LIN {X 0,Y 516.172,Z 433.767,A -85,B 0,C 180,E1 -4909.681,E2 -4909.681} C_VEL
LIN {X 0,Y 516.191,Z 433.561,A -85,B 0,C 180,E1 -4910.899,E2 -4910.899} C_VEL
LIN {X 0,Y 516.175,Z 431.928,A -85,B 0,C 180,E1 -4912.214,E2 -4912.214} C_VEL
LIN {X 0,Y 516.288,Z 429.068,A -85,B 0,C 180,E1 -4913.429,E2 -4913.429} C_VEL
LIN {X 0,Y 516.355,Z 425.479,A -85,B 0,C 180,E1 -4914.491,E2 -4914.491} C_VEL
LIN {X 0,Y 516.462,Z 420.419,A -85,B 0,C 180,E1 -4915.616,E2 -4915.616} C_VEL
LIN {X 0,Y 516.626,Z 413.305,A -85,B 0,C 180,E1 -4916.803,E2 -4916.803} C_VEL
LIN {X 0,Y 516.784,Z 406.191,A -85,B 0,C 180,E1 -4917.726,E2 -4917.726} C_VEL
LIN {X 0,Y 516.968,Z 399.489,A -85,B 0,C 180,E1 -4918.439,E2 -4918.439} C_VEL
LIN {X 0,Y 517.059,Z 393.49,A -85,B 0,C 180,E1 -4918.98,E2 -4918.98} C_VEL
LIN {X 0,Y 517.216,Z 385.286,A -85,B 0,C 180,E1 -4919.591,E2 -4919.591} C_VEL
LIN {X 0,Y 517.396,Z 376.875,A -85,B 0,C 180,E1 -4920.093,E2 -4920.093} C_VEL
LIN {X 0,Y 517.533,Z 368.879,A -85,B 0,C 180,E1 -4920.47,E2 -4920.47} C_VEL
LIN {X 0,Y 517.4,Z 363.16,A -85,B 0,C 180,E1 -4920.698,E2 -4920.698} C_VEL
LIN {X 0,Y 516.294,Z 355.849,A -85,B 0,C 180,E1 -4920.963,E2 -4920.963} C_VEL
LIN {X 0,Y 516.339,Z 351.268,A -85,B 0,C 180,E1 -4924.178,E2 -4924.178} C_VEL
LIN {X 0,Y 516.335,Z 347.701,A -85,B 0,C 180,E1 -4926.75,E2 -4926.75} C_VEL
LIN {X 0,Y 516.376,Z 343.028,A -85,B 0,C 180,E1 -4930.107,E2 -4930.107} C_VEL
LIN {X 0,Y 516.437,Z 339.664,A -85,B 0,C 180,E1 -4932.578,E2 -4932.578} C_VEL
LIN {X 0,Y 516.461,Z 335.27,A -85,B 0,C 180,E1 -4935.821,E2 -4935.821} C_VEL
LIN {X 0,Y 516.631,Z 330.958,A -85,B 0,C 180,E1 -4939.02,E2 -4939.02} C_VEL
LIN {X 0,Y 516.634,Z 328.948,A -85,B 0,C 180,E1 -4940.604,E2 -4940.604} C_VEL
LIN {X 0,Y 517.004,Z 328.898,A -85,B 0,C 180,E1 -4942.972,E2 -4942.972} C_VEL
LIN {X 0,Y 516.928,Z 328.907,A -85,B 0,C 180,E1 -4945.32,E2 -4945.32} C_VEL
LIN {X 0,Y 517.072,Z 328.89,A -85,B 0,C 180,E1 -4947.662,E2 -4947.662} C_VEL
LIN {X 0,Y 517.085,Z 328.89,A -85,B 0,C 180,E1 -4950.778,E2 -4950.778} C_VEL
LIN {X 0,Y 517.006,Z 328.899,A -85,B 0,C 180,E1 -4953.116,E2 -4953.116} C_VEL
LIN {X 0,Y 517,Z 328.899,A -85,B 0,C 180,E1 -4956.242,E2 -4956.242} C_VEL
LIN {X 0,Y 516.948,Z 328.907,A -85,B 0,C 180,E1 -4959.388,E2 -4959.388} C_VEL
LIN {X 0,Y 516.971,Z 328.905,A -85,B 0,C 180,E1 -4961.823,E2 -4961.823} C_VEL
LIN {X 0,Y 516.931,Z 328.907,A -85,B 0,C 180,E1 -4965.146,E2 -4965.146} C_VEL
LIN {X 0,Y 516.913,Z 328.909,A -85,B 0,C 180,E1 -4968.221,E2 -4968.221} C_VEL
LIN {X 0,Y 516.9,Z 328.911,A -85,B 0,C 180,E1 -4970.701,E2 -4970.701} C_VEL
LIN {X 0,Y 516.897,Z 328.912,A -85,B 0,C 180,E1 -4974.071,E2 -4974.071} C_VEL
LIN {X 0,Y 516.915,Z 328.91,A -85,B 0,C 180,E1 -4976.657,E2 -4976.657} C_VEL
LIN {X 0,Y 516.91,Z 328.911,A -85,B 0,C 180,E1 -4979.526,E2 -4979.526} C_VEL
LIN {X 0,Y 516.887,Z 328.914,A -85,B 0,C 180,E1 -4982.544,E2 -4982.544} C_VEL
LIN {X 0,Y 516.87,Z 328.915,A -85,B 0,C 180,E1 -4985.332,E2 -4985.332} C_VEL
LIN {X 0,Y 516.87,Z 328.915,A -85,B 0,C 180,E1 -4987.944,E2 -4987.944} C_VEL
LIN {X 0,Y 516.893,Z 328.913,A -85,B 0,C 180,E1 -4990.739,E2 -4990.739} C_VEL
LIN {X 0,Y 516.868,Z 328.914,A -85,B 0,C 180,E1 -4993.903,E2 -4993.903} C_VEL
LIN {X 0,Y 516.867,Z 328.915,A -85,B 0,C 180,E1 -4996.107,E2 -4996.107} C_VEL
LIN {X 0,Y 516.889,Z 328.915,A -85,B 0,C 180,E1 -4999.26,E2 -4999.26} C_VEL
LIN {X 0,Y 516.871,Z 328.916,A -85,B 0,C 180,E1 -5002.056,E2 -5002.056} C_VEL
LIN {X 0,Y 516.882,Z 328.915,A -85,B 0,C 180,E1 -5005.177,E2 -5005.177} C_VEL
LIN {X 0,Y 516.869,Z 328.917,A -85,B 0,C 180,E1 -5007.976,E2 -5007.976} C_VEL
LIN {X 0,Y 516.922,Z 328.909,A -85,B 0,C 180,E1 -5010.697,E2 -5010.697} C_VEL
LIN {X 0,Y 516.928,Z 328.908,A -85,B 0,C 180,E1 -5013.804,E2 -5013.804} C_VEL
LIN {X 0,Y 516.885,Z 328.913,A -85,B 0,C 180,E1 -5016.778,E2 -5016.778} C_VEL
LIN {X 0,Y 516.926,Z 328.907,A -85,B 0,C 180,E1 -5019.732,E2 -5019.732} C_VEL
LIN {X 0,Y 516.918,Z 328.91,A -85,B 0,C 180,E1 -5022.597,E2 -5022.597} C_VEL
LIN {X 0,Y 516.928,Z 328.908,A -85,B 0,C 180,E1 -5025.031,E2 -5025.031} C_VEL
LIN {X 0,Y 516.991,Z 328.901,A -85,B 0,C 180,E1 -5028.235,E2 -5028.235} C_VEL
LIN {X 0,Y 516.96,Z 328.904,A -85,B 0,C 180,E1 -5031.4,E2 -5031.4} C_VEL
LIN {X 0,Y 517,Z 328.9,A -85,B 0,C 180,E1 -5033.758,E2 -5033.758} C_VEL
LIN {X 0,Y 517.076,Z 328.889,A -85,B 0,C 180,E1 -5037.664,E2 -5037.664} C_VEL
LIN {X 0,Y 517.087,Z 328.889,A -85,B 0,C 180,E1 -5040.78,E2 -5040.78} C_VEL
LIN {X 0,Y 517.007,Z 328.899,A -85,B 0,C 180,E1 -5043.118,E2 -5043.118} C_VEL
LIN {X 0,Y 517,Z 328.899,A -85,B 0,C 180,E1 -5046.244,E2 -5046.244} C_VEL
LIN {X 0,Y 516.945,Z 328.907,A -85,B 0,C 180,E1 -5049.39,E2 -5049.39} C_VEL
LIN {X 0,Y 516.973,Z 328.903,A -85,B 0,C 180,E1 -5051.825,E2 -5051.825} C_VEL
LIN {X 0,Y 516.934,Z 328.908,A -85,B 0,C 180,E1 -5055.147,E2 -5055.147} C_VEL
LIN {X 0,Y 516.917,Z 328.908,A -85,B 0,C 180,E1 -5058.223,E2 -5058.223} C_VEL
LIN {X 0,Y 516.903,Z 328.91,A -85,B 0,C 180,E1 -5060.702,E2 -5060.702} C_VEL
LIN {X 0,Y 516.903,Z 328.91,A -85,B 0,C 180,E1 -5064.073,E2 -5064.073} C_VEL
LIN {X 0,Y 516.921,Z 328.908,A -85,B 0,C 180,E1 -5066.659,E2 -5066.659} C_VEL
LIN {X 0,Y 516.917,Z 328.91,A -85,B 0,C 180,E1 -5069.528,E2 -5069.528} C_VEL
LIN {X 0,Y 516.89,Z 328.913,A -85,B 0,C 180,E1 -5072.545,E2 -5072.545} C_VEL
LIN {X 0,Y 516.877,Z 328.914,A -85,B 0,C 180,E1 -5075.334,E2 -5075.334} C_VEL
LIN {X 0,Y 516.875,Z 328.914,A -85,B 0,C 180,E1 -5077.945,E2 -5077.945} C_VEL
LIN {X 0,Y 516.879,Z 328.916,A -85,B 0,C 180,E1 -5080.743,E2 -5080.743} C_VEL
LIN {X 0,Y 516.898,Z 328.912,A -85,B 0,C 180,E1 -5082.83,E2 -5082.83} C_VEL
LIN {X 0,Y 516.917,Z 328.909,A -85,B 0,C 180,E1 -5085.011,E2 -5085.011} C_VEL
LIN {X 0,Y 516.912,Z 328.91,A -85,B 0,C 180,E1 -5088.399,E2 -5088.399} C_VEL
LIN {X 0,Y 516.878,Z 328.914,A -85,B 0,C 180,E1 -5091.286,E2 -5091.286} C_VEL
LIN {X 0,Y 516.912,Z 328.911,A -85,B 0,C 180,E1 -5094.664,E2 -5094.664} C_VEL
LIN {X 0,Y 516.971,Z 329.042,A -85,B 0,C 180,E1 -5095.089,E2 -5095.089} C_VEL
LIN {X 0,Y 517.728,Z 334.233,A -85,B 0,C 180,E1 -5097.114,E2 -5097.114} C_VEL
LIN {X 0,Y 517.54,Z 340.461,A -85,B 0,C 180,E1 -5099.389,E2 -5099.389} C_VEL
LIN {X 0,Y 517.319,Z 347.853,A -85,B 0,C 180,E1 -5102.013,E2 -5102.013} C_VEL
LIN {X 0,Y 517.105,Z 355.534,A -85,B 0,C 180,E1 -5104.653,E2 -5104.653} C_VEL
LIN {X 0,Y 516.938,Z 363.131,A -85,B 0,C 180,E1 -5107.205,E2 -5107.205} C_VEL
LIN {X 0,Y 516.741,Z 373.276,A -85,B 0,C 180,E1 -5110.537,E2 -5110.537} C_VEL
LIN {X 0,Y 516.594,Z 382.323,A -85,B 0,C 180,E1 -5113.401,E2 -5113.401} C_VEL
LIN {X 0,Y 516.522,Z 390.164,A -85,B 0,C 180,E1 -5115.824,E2 -5115.824} C_VEL
LIN {X 0,Y 516.441,Z 398.672,A -85,B 0,C 180,E1 -5118.469,E2 -5118.469} C_VEL
LIN {X 0,Y 516.417,Z 400.594,A -85,B 0,C 180,E1 -5119.042,E2 -5119.042} C_VEL
LIN {X 0,Y 517.546,Z 412.161,A -85,B 0,C 180,E1 -5119.388,E2 -5119.388} C_VEL
LIN {X 0,Y 517.385,Z 422.491,A -85,B 0,C 180,E1 -5119.83,E2 -5119.83} C_VEL
LIN {X 0,Y 517.179,Z 431.229,A -85,B 0,C 180,E1 -5120.32,E2 -5120.32} C_VEL
LIN {X 0,Y 517.022,Z 439.578,A -85,B 0,C 180,E1 -5120.909,E2 -5120.909} C_VEL
LIN {X 0,Y 516.818,Z 447.479,A -85,B 0,C 180,E1 -5121.595,E2 -5121.595} C_VEL
LIN {X 0,Y 516.672,Z 454.871,A -85,B 0,C 180,E1 -5122.38,E2 -5122.38} C_VEL
LIN {X 0,Y 516.533,Z 462.212,A -85,B 0,C 180,E1 -5123.337,E2 -5123.337} C_VEL
LIN {X 0,Y 516.448,Z 468.264,A -85,B 0,C 180,E1 -5124.339,E2 -5124.339} C_VEL
LIN {X 0,Y 516.314,Z 472.898,A -85,B 0,C 180,E1 -5125.316,E2 -5125.316} C_VEL
LIN {X 0,Y 516.364,Z 475.915,A -85,B 0,C 180,E1 -5126.099,E2 -5126.099} C_VEL
LIN {X 0,Y 516.294,Z 478.248,A -85,B 0,C 180,E1 -5126.88,E2 -5126.88} C_VEL
LIN {X 0,Y 516.263,Z 480.005,A -85,B 0,C 180,E1 -5127.66,E2 -5127.66} C_VEL
LIN {X 0,Y 516.191,Z 481.261,A -85,B 0,C 180,E1 -5128.441,E2 -5128.441} C_VEL
LIN {X 0,Y 516.158,Z 482.041,A -85,B 0,C 180,E1 -5129.221,E2 -5129.221} C_VEL
LIN {X 0,Y 516.156,Z 482.335,A -85,B 0,C 180,E1 -5130.001,E2 -5130.001} C_VEL
LIN {X 0,Y 516.158,Z 482.036,A -85,B 0,C 180,E1 -5130.781,E2 -5130.781} C_VEL
LIN {X 0,Y 516.191,Z 481.25,A -85,B 0,C 180,E1 -5131.561,E2 -5131.561} C_VEL
LIN {X 0,Y 516.263,Z 479.988,A -85,B 0,C 180,E1 -5132.342,E2 -5132.342} C_VEL
LIN {X 0,Y 516.323,Z 477.065,A -85,B 0,C 180,E1 -5133.513,E2 -5133.513} C_VEL
LIN {X 0,Y 516.342,Z 474.398,A -85,B 0,C 180,E1 -5134.294,E2 -5134.294} C_VEL
LIN {X 0,Y 516.425,Z 469.184,A -85,B 0,C 180,E1 -5135.467,E2 -5135.467} C_VEL
LIN {X 0,Y 516.516,Z 463.713,A -85,B 0,C 180,E1 -5136.423,E2 -5136.423} C_VEL
LIN {X 0,Y 516.633,Z 456.509,A -85,B 0,C 180,E1 -5137.426,E2 -5137.426} C_VEL
LIN {X 0,Y 516.797,Z 448.426,A -85,B 0,C 180,E1 -5138.309,E2 -5138.309} C_VEL
LIN {X 0,Y 516.989,Z 440.714,A -85,B 0,C 180,E1 -5138.995,E2 -5138.995} C_VEL
LIN {X 0,Y 517.146,Z 432.616,A -85,B 0,C 180,E1 -5139.584,E2 -5139.584} C_VEL
LIN {X 0,Y 517.337,Z 424.231,A -85,B 0,C 180,E1 -5140.074,E2 -5140.074} C_VEL
LIN {X 0,Y 517.514,Z 415.677,A -85,B 0,C 180,E1 -5140.466,E2 -5140.466} C_VEL
LIN {X 0,Y 517.365,Z 408.802,A -85,B 0,C 180,E1 -5140.717,E2 -5140.717} C_VEL
LIN {X 0,Y 516.427,Z 400.26,A -85,B 0,C 180,E1 -5140.984,E2 -5140.984} C_VEL
LIN {X 0,Y 516.52,Z 389.965,A -85,B 0,C 180,E1 -5144.178,E2 -5144.178} C_VEL
LIN {X 0,Y 516.594,Z 380.776,A -85,B 0,C 180,E1 -5147.008,E2 -5147.008} C_VEL
LIN {X 0,Y 516.734,Z 373.032,A -85,B 0,C 180,E1 -5149.465,E2 -5149.465} C_VEL
LIN {X 0,Y 516.868,Z 364.07,A -85,B 0,C 180,E1 -5152.389,E2 -5152.389} C_VEL
LIN {X 0,Y 517.089,Z 355.16,A -85,B 0,C 180,E1 -5155.35,E2 -5155.35} C_VEL
LIN {X 0,Y 517.301,Z 346.385,A -85,B 0,C 180,E1 -5158.393,E2 -5158.393} C_VEL
LIN {X 0,Y 517.626,Z 338.595,A -85,B 0,C 180,E1 -5161.198,E2 -5161.198} C_VEL
LIN {X 0,Y 517.721,Z 334.128,A -85,B 0,C 180,E1 -5162.889,E2 -5162.889} C_VEL
LIN {X 0,Y 516.897,Z 328.913,A -85,B 0,C 180,E1 -5165.01,E2 -5165.01} C_VEL
LIN {X 0,Y 516.885,Z 328.915,A -85,B 0,C 180,E1 -5167.943,E2 -5167.943} C_VEL
LIN {X 0,Y 516.888,Z 328.918,A -85,B 0,C 180,E1 -5170.742,E2 -5170.742} C_VEL
LIN {X 0,Y 516.89,Z 328.918,A -85,B 0,C 180,E1 -5172.832,E2 -5172.832} C_VEL
LIN {X 0,Y 516.901,Z 328.915,A -85,B 0,C 180,E1 -5175.007,E2 -5175.007} C_VEL
LIN {X 0,Y 516.919,Z 328.91,A -85,B 0,C 180,E1 -5178.399,E2 -5178.399} C_VEL
LIN {X 0,Y 516.883,Z 328.915,A -85,B 0,C 180,E1 -5181.284,E2 -5181.284} C_VEL
LIN {X 0,Y 516.877,Z 328.914,A -85,B 0,C 180,E1 -5184.22,E2 -5184.22} C_VEL
LIN {X 0,Y 516.887,Z 328.915,A -85,B 0,C 180,E1 -5187.052,E2 -5187.052} C_VEL
LIN {X 0,Y 516.893,Z 328.912,A -85,B 0,C 180,E1 -5189.796,E2 -5189.796} C_VEL
LIN {X 0,Y 516.93,Z 328.907,A -85,B 0,C 180,E1 -5192.467,E2 -5192.467} C_VEL
LIN {X 0,Y 516.915,Z 328.911,A -85,B 0,C 180,E1 -5195.072,E2 -5195.072} C_VEL
LIN {X 0,Y 516.892,Z 328.912,A -85,B 0,C 180,E1 -5198.462,E2 -5198.462} C_VEL
LIN {X 0,Y 516.906,Z 328.912,A -85,B 0,C 180,E1 -5200.954,E2 -5200.954} C_VEL
LIN {X 0,Y 516.911,Z 328.911,A -85,B 0,C 180,E1 -5203.41,E2 -5203.41} C_VEL
LIN {X 0,Y 516.898,Z 328.914,A -85,B 0,C 180,E1 -5205.833,E2 -5205.833} C_VEL
LIN {X 0,Y 516.973,Z 328.905,A -85,B 0,C 180,E1 -5208.233,E2 -5208.233} C_VEL
LIN {X 0,Y 516.961,Z 328.904,A -85,B 0,C 180,E1 -5211.399,E2 -5211.399} C_VEL
LIN {X 0,Y 517.029,Z 328.896,A -85,B 0,C 180,E1 -5214.539,E2 -5214.539} C_VEL
LIN {X 0,Y 517.084,Z 328.891,A -85,B 0,C 180,E1 -5217.662,E2 -5217.662} C_VEL
LIN {X 0,Y 517.099,Z 328.886,A -85,B 0,C 180,E1 -5220.778,E2 -5220.778} C_VEL
LIN {X 0,Y 517.014,Z 328.897,A -85,B 0,C 180,E1 -5223.116,E2 -5223.116} C_VEL
LIN {X 0,Y 517.014,Z 328.898,A -85,B 0,C 180,E1 -5226.242,E2 -5226.242} C_VEL
LIN {X 0,Y 516.944,Z 328.908,A -85,B 0,C 180,E1 -5229.389,E2 -5229.389} C_VEL
LIN {X 0,Y 516.956,Z 328.907,A -85,B 0,C 180,E1 -5231.806,E2 -5231.806} C_VEL
LIN {X 0,Y 516.948,Z 328.908,A -85,B 0,C 180,E1 -5235.145,E2 -5235.145} C_VEL
LIN {X 0,Y 516.852,Z 328.921,A -85,B 0,C 180,E1 -5237.853,E2 -5237.853} C_VEL
LIN {X 0,Y 516.655,Z 328.945,A -85,B 0,C 180,E1 -5239.054,E2 -5239.054} C_VEL
LIN {X 0,Y 516.57,Z 332.084,A -85,B 0,C 180,E1 -5241.55,E2 -5241.55} C_VEL
LIN {X 0,Y 516.545,Z 335.708,A -85,B 0,C 180,E1 -5244.273,E2 -5244.273} C_VEL
LIN {X 0,Y 516.45,Z 338.912,A -85,B 0,C 180,E1 -5246.683,E2 -5246.683} C_VEL
LIN {X 0,Y 516.427,Z 342.589,A -85,B 0,C 180,E1 -5249.428,E2 -5249.428} C_VEL
LIN {X 0,Y 516.338,Z 346.763,A -85,B 0,C 180,E1 -5252.445,E2 -5252.445} C_VEL
LIN {X 0,Y 516.314,Z 350.521,A -85,B 0,C 180,E1 -5255.242,E2 -5255.242} C_VEL
LIN {X 0,Y 516.235,Z 354.157,A -85,B 0,C 180,E1 -5257.85,E2 -5257.85} C_VEL
LIN {X 0,Y 516.279,Z 356.115,A -85,B 0,C 180,E1 -5259.153,E2 -5259.153} C_VEL
LIN {X 0,Y 517.638,Z 366.34,A -85,B 0,C 180,E1 -5259.513,E2 -5259.513} C_VEL
LIN {X 0,Y 517.445,Z 375.523,A -85,B 0,C 180,E1 -5259.921,E2 -5259.921} C_VEL
LIN {X 0,Y 517.305,Z 383.809,A -85,B 0,C 180,E1 -5260.397,E2 -5260.397} C_VEL
LIN {X 0,Y 517.089,Z 391.927,A -85,B 0,C 180,E1 -5260.978,E2 -5260.978} C_VEL
LIN {X 0,Y 516.973,Z 399.12,A -85,B 0,C 180,E1 -5261.608,E2 -5261.608} C_VEL
LIN {X 0,Y 516.816,Z 405.767,A -85,B 0,C 180,E1 -5262.308,E2 -5262.308} C_VEL
LIN {X 0,Y 516.68,Z 411.965,A -85,B 0,C 180,E1 -5263.094,E2 -5263.094} C_VEL
LIN {X 0,Y 516.499,Z 418.569,A -85,B 0,C 180,E1 -5264.126,E2 -5264.126} C_VEL
LIN {X 0,Y 515.834,Z 421.674,A -85,B 0,C 180,E1 -5264.679,E2 -5264.679} C_VEL
LIN {X 0,Y 514.218,Z 424.431,A -85,B 0,C 180,E1 -5265.238,E2 -5265.238} C_VEL
LIN {X 0,Y 510.396,Z 428.868,A -85,B 0,C 180,E1 -5266.404,E2 -5266.404} C_VEL
LIN {X 0,Y 509.222,Z 430.843,A -85,B 0,C 180,E1 -5267.14,E2 -5267.14} C_VEL
LIN {X 0,Y 509.192,Z 431.048,A -85,B 0,C 180,E1 -5267.248,E2 -5267.248} C_VEL
LIN {X 0,Y 509.139,Z 433.208,A -85,B 0,C 180,E1 -5268.502,E2 -5268.502} C_VEL
LIN {X 0,Y 509.102,Z 434.048,A -85,B 0,C 180,E1 -5269.546,E2 -5269.546} C_VEL
LIN {X 0,Y 509.084,Z 434.009,A -85,B 0,C 180,E1 -5270.63,E2 -5270.63} C_VEL
LIN {X 0,Y 509.092,Z 432.825,A -85,B 0,C 180,E1 -5271.893,E2 -5271.893} C_VEL
LIN {X 0,Y 509.179,Z 430.248,A -85,B 0,C 180,E1 -5273.181,E2 -5273.181} C_VEL
LIN {X 0,Y 509.275,Z 427.574,A -85,B 0,C 180,E1 -5274.084,E2 -5274.084} C_VEL
LIN {X 0,Y 509.334,Z 422.599,A -85,B 0,C 180,E1 -5275.306,E2 -5275.306} C_VEL
LIN {X 0,Y 509.439,Z 418.025,A -85,B 0,C 180,E1 -5276.187,E2 -5276.187} C_VEL
LIN {X 0,Y 509.572,Z 413.446,A -85,B 0,C 180,E1 -5276.921,E2 -5276.921} C_VEL
LIN {X 0,Y 509.771,Z 406.566,A -85,B 0,C 180,E1 -5277.824,E2 -5277.824} C_VEL
LIN {X 0,Y 509.971,Z 399.395,A -85,B 0,C 180,E1 -5278.594,E2 -5278.594} C_VEL
LIN {X 0,Y 510.072,Z 392.071,A -85,B 0,C 180,E1 -5279.244,E2 -5279.244} C_VEL
LIN {X 0,Y 510.308,Z 382.77,A -85,B 0,C 180,E1 -5279.91,E2 -5279.91} C_VEL
LIN {X 0,Y 510.566,Z 371.407,A -85,B 0,C 180,E1 -5280.52,E2 -5280.52} C_VEL
LIN {X 0,Y 510.369,Z 363.419,A -85,B 0,C 180,E1 -5280.847,E2 -5280.847} C_VEL
LIN {X 0,Y 509.201,Z 356.154,A -85,B 0,C 180,E1 -5281.113,E2 -5281.113} C_VEL
LIN {X 0,Y 509.25,Z 352.367,A -85,B 0,C 180,E1 -5283.792,E2 -5283.792} C_VEL
LIN {X 0,Y 509.245,Z 348.725,A -85,B 0,C 180,E1 -5286.407,E2 -5286.407} C_VEL
LIN {X 0,Y 509.249,Z 345.203,A -85,B 0,C 180,E1 -5288.971,E2 -5288.971} C_VEL
LIN {X 0,Y 509.391,Z 340.63,A -85,B 0,C 180,E1 -5292.329,E2 -5292.329} C_VEL
LIN {X 0,Y 509.407,Z 336.179,A -85,B 0,C 180,E1 -5295.62,E2 -5295.62} C_VEL
LIN {X 0,Y 509.559,Z 331.841,A -85,B 0,C 180,E1 -5298.866,E2 -5298.866} C_VEL
LIN {X 0,Y 509.57,Z 329.827,A -85,B 0,C 180,E1 -5300.473,E2 -5300.473} C_VEL
LIN {X 0,Y 509.942,Z 329.778,A -85,B 0,C 180,E1 -5302.874,E2 -5302.874} C_VEL
LIN {X 0,Y 509.896,Z 329.783,A -85,B 0,C 180,E1 -5305.255,E2 -5305.255} C_VEL
LIN {X 0,Y 510.044,Z 329.766,A -85,B 0,C 180,E1 -5307.63,E2 -5307.63} C_VEL
LIN {X 0,Y 510.044,Z 329.766,A -85,B 0,C 180,E1 -5309.999,E2 -5309.999} C_VEL
LIN {X 0,Y 510.047,Z 329.765,A -85,B 0,C 180,E1 -5312.368,E2 -5312.368} C_VEL
LIN {X 0,Y 509.998,Z 329.772,A -85,B 0,C 180,E1 -5315.534,E2 -5315.534} C_VEL
LIN {X 0,Y 509.941,Z 329.78,A -85,B 0,C 180,E1 -5317.921,E2 -5317.921} C_VEL
LIN {X 0,Y 509.914,Z 329.781,A -85,B 0,C 180,E1 -5321.124,E2 -5321.124} C_VEL
LIN {X 0,Y 509.852,Z 329.789,A -85,B 0,C 180,E1 -5324.365,E2 -5324.365} C_VEL
LIN {X 0,Y 509.89,Z 329.786,A -85,B 0,C 180,E1 -5327.651,E2 -5327.651} C_VEL
LIN {X 0,Y 509.873,Z 329.787,A -85,B 0,C 180,E1 -5330.401,E2 -5330.401} C_VEL
LIN {X 0,Y 509.823,Z 329.794,A -85,B 0,C 180,E1 -5333.562,E2 -5333.562} C_VEL
LIN {X 0,Y 509.899,Z 329.784,A -85,B 0,C 180,E1 -5336.379,E2 -5336.379} C_VEL
LIN {X 0,Y 509.872,Z 329.789,A -85,B 0,C 180,E1 -5338.843,E2 -5338.843} C_VEL
LIN {X 0,Y 509.812,Z 329.794,A -85,B 0,C 180,E1 -5341.589,E2 -5341.589} C_VEL
LIN {X 0,Y 509.84,Z 329.79,A -85,B 0,C 180,E1 -5344.413,E2 -5344.413} C_VEL
LIN {X 0,Y 509.808,Z 329.797,A -85,B 0,C 180,E1 -5347.34,E2 -5347.34} C_VEL
LIN {X 0,Y 509.848,Z 329.789,A -85,B 0,C 180,E1 -5350.38,E2 -5350.38} C_VEL
LIN {X 0,Y 509.826,Z 329.794,A -85,B 0,C 180,E1 -5353.064,E2 -5353.064} C_VEL
LIN {X 0,Y 509.815,Z 329.795,A -85,B 0,C 180,E1 -5355.792,E2 -5355.792} C_VEL
LIN {X 0,Y 509.85,Z 329.79,A -85,B 0,C 180,E1 -5358.576,E2 -5358.576} C_VEL
LIN {X 0,Y 509.843,Z 329.791,A -85,B 0,C 180,E1 -5361.785,E2 -5361.785} C_VEL
LIN {X 0,Y 509.833,Z 329.792,A -85,B 0,C 180,E1 -5364.624,E2 -5364.624} C_VEL
LIN {X 0,Y 509.852,Z 329.789,A -85,B 0,C 180,E1 -5367.482,E2 -5367.482} C_VEL
LIN {X 0,Y 509.867,Z 329.789,A -85,B 0,C 180,E1 -5370.269,E2 -5370.269} C_VEL
LIN {X 0,Y 509.871,Z 329.788,A -85,B 0,C 180,E1 -5372.945,E2 -5372.945} C_VEL
LIN {X 0,Y 509.875,Z 329.786,A -85,B 0,C 180,E1 -5375.575,E2 -5375.575} C_VEL
LIN {X 0,Y 509.836,Z 329.791,A -85,B 0,C 180,E1 -5378.15,E2 -5378.15} C_VEL
LIN {X 0,Y 509.852,Z 329.789,A -85,B 0,C 180,E1 -5380.682,E2 -5380.682} C_VEL
LIN {X 0,Y 509.875,Z 329.786,A -85,B 0,C 180,E1 -5383.175,E2 -5383.175} C_VEL
LIN {X 0,Y 509.851,Z 329.788,A -85,B 0,C 180,E1 -5385.635,E2 -5385.635} C_VEL
LIN {X 0,Y 509.91,Z 329.781,A -85,B 0,C 180,E1 -5388.875,E2 -5388.875} C_VEL
LIN {X 0,Y 509.94,Z 329.78,A -85,B 0,C 180,E1 -5392.079,E2 -5392.079} C_VEL
LIN {X 0,Y 509.973,Z 329.777,A -85,B 0,C 180,E1 -5394.465,E2 -5394.465} C_VEL
LIN {X 0,Y 510.047,Z 329.765,A -85,B 0,C 180,E1 -5397.632,E2 -5397.632} C_VEL
LIN {X 0,Y 510.056,Z 329.764,A -85,B 0,C 180,E1 -5400.79,E2 -5400.79} C_VEL
LIN {X 0,Y 509.95,Z 329.778,A -85,B 0,C 180,E1 -5403.161,E2 -5403.161} C_VEL
LIN {X 0,Y 509.968,Z 329.775,A -85,B 0,C 180,E1 -5406.33,E2 -5406.33} C_VEL
LIN {X 0,Y 509.906,Z 329.782,A -85,B 0,C 180,E1 -5408.721,E2 -5408.721} C_VEL
LIN {X 0,Y 509.941,Z 329.779,A -85,B 0,C 180,E1 -5411.931,E2 -5411.931} C_VEL
LIN {X 0,Y 509.884,Z 329.787,A -85,B 0,C 180,E1 -5415.243,E2 -5415.243} C_VEL
LIN {X 0,Y 509.879,Z 329.786,A -85,B 0,C 180,E1 -5418.002,E2 -5418.002} C_VEL
LIN {X 0,Y 509.841,Z 329.791,A -85,B 0,C 180,E1 -5421.003,E2 -5421.003} C_VEL
LIN {X 0,Y 509.828,Z 329.794,A -85,B 0,C 180,E1 -5423.564,E2 -5423.564} C_VEL
LIN {X 0,Y 509.905,Z 329.783,A -85,B 0,C 180,E1 -5426.38,E2 -5426.38} C_VEL
LIN {X 0,Y 509.878,Z 329.788,A -85,B 0,C 180,E1 -5428.845,E2 -5428.845} C_VEL
LIN {X 0,Y 509.814,Z 329.794,A -85,B 0,C 180,E1 -5431.591,E2 -5431.591} C_VEL
LIN {X 0,Y 509.848,Z 329.789,A -85,B 0,C 180,E1 -5434.414,E2 -5434.414} C_VEL
LIN {X 0,Y 509.812,Z 329.795,A -85,B 0,C 180,E1 -5437.342,E2 -5437.342} C_VEL
LIN {X 0,Y 509.832,Z 329.791,A -85,B 0,C 180,E1 -5440.383,E2 -5440.383} C_VEL
LIN {X 0,Y 509.834,Z 329.794,A -85,B 0,C 180,E1 -5443.065,E2 -5443.065} C_VEL
LIN {X 0,Y 509.825,Z 329.793,A -85,B 0,C 180,E1 -5445.793,E2 -5445.793} C_VEL
LIN {X 0,Y 509.853,Z 329.789,A -85,B 0,C 180,E1 -5448.576,E2 -5448.576} C_VEL
LIN {X 0,Y 509.847,Z 329.791,A -85,B 0,C 180,E1 -5451.788,E2 -5451.788} C_VEL
LIN {X 0,Y 509.927,Z 329.836,A -85,B 0,C 180,E1 -5454.873,E2 -5454.873} C_VEL
LIN {X 0,Y 510.74,Z 335.397,A -85,B 0,C 180,E1 -5457.076,E2 -5457.076} C_VEL
LIN {X 0,Y 510.613,Z 340.498,A -85,B 0,C 180,E1 -5458.976,E2 -5458.976} C_VEL
LIN {X 0,Y 510.297,Z 349.099,A -85,B 0,C 180,E1 -5462.08,E2 -5462.08} C_VEL
LIN {X 0,Y 510.018,Z 357.82,A -85,B 0,C 180,E1 -5465.12,E2 -5465.12} C_VEL
LIN {X 0,Y 509.838,Z 365.73,A -85,B 0,C 180,E1 -5467.798,E2 -5467.798} C_VEL
LIN {X 0,Y 509.66,Z 374.379,A -85,B 0,C 180,E1 -5470.675,E2 -5470.675} C_VEL
LIN {X 0,Y 509.518,Z 383.403,A -85,B 0,C 180,E1 -5473.576,E2 -5473.576} C_VEL
LIN {X 0,Y 509.439,Z 391.202,A -85,B 0,C 180,E1 -5476.031,E2 -5476.031} C_VEL
LIN {X 0,Y 509.348,Z 400.224,A -85,B 0,C 180,E1 -5478.888,E2 -5478.888} C_VEL
LIN {X 0,Y 510.55,Z 411.809,A -85,B 0,C 180,E1 -5479.241,E2 -5479.241} C_VEL
LIN {X 0,Y 510.38,Z 422.144,A -85,B 0,C 180,E1 -5479.689,E2 -5479.689} C_VEL
LIN {X 0,Y 510.171,Z 430.884,A -85,B 0,C 180,E1 -5480.186,E2 -5480.186} C_VEL
LIN {X 0,Y 509.993,Z 439.235,A -85,B 0,C 180,E1 -5480.783,E2 -5480.783} C_VEL
LIN {X 0,Y 509.791,Z 447.139,A -85,B 0,C 180,E1 -5481.478,E2 -5481.478} C_VEL
LIN {X 0,Y 509.605,Z 454.531,A -85,B 0,C 180,E1 -5482.274,E2 -5482.274} C_VEL
LIN {X 0,Y 509.433,Z 462.658,A -85,B 0,C 180,E1 -5483.361,E2 -5483.361} C_VEL
LIN {X 0,Y 509.341,Z 468.894,A -85,B 0,C 180,E1 -5484.458,E2 -5484.458} C_VEL
LIN {X 0,Y 509.238,Z 474.096,A -85,B 0,C 180,E1 -5485.648,E2 -5485.648} C_VEL
LIN {X 0,Y 509.245,Z 476.759,A -85,B 0,C 180,E1 -5486.44,E2 -5486.44} C_VEL
LIN {X 0,Y 509.192,Z 479.675,A -85,B 0,C 180,E1 -5487.628,E2 -5487.628} C_VEL
LIN {X 0,Y 509.111,Z 480.93,A -85,B 0,C 180,E1 -5488.419,E2 -5488.419} C_VEL
LIN {X 0,Y 509.071,Z 481.71,A -85,B 0,C 180,E1 -5489.21,E2 -5489.21} C_VEL
LIN {X 0,Y 509.067,Z 482.003,A -85,B 0,C 180,E1 -5490.001,E2 -5490.001} C_VEL
LIN {X 0,Y 509.071,Z 481.703,A -85,B 0,C 180,E1 -5490.792,E2 -5490.792} C_VEL
LIN {X 0,Y 509.111,Z 480.916,A -85,B 0,C 180,E1 -5491.583,E2 -5491.583} C_VEL
LIN {X 0,Y 509.192,Z 479.652,A -85,B 0,C 180,E1 -5492.374,E2 -5492.374} C_VEL
LIN {X 0,Y 509.243,Z 476.726,A -85,B 0,C 180,E1 -5493.562,E2 -5493.562} C_VEL
LIN {X 0,Y 509.237,Z 474.053,A -85,B 0,C 180,E1 -5494.354,E2 -5494.354} C_VEL
LIN {X 0,Y 509.342,Z 468.834,A -85,B 0,C 180,E1 -5495.544,E2 -5495.544} C_VEL
LIN {X 0,Y 509.438,Z 462.562,A -85,B 0,C 180,E1 -5496.644,E2 -5496.644} C_VEL
LIN {X 0,Y 509.607,Z 454.44,A -85,B 0,C 180,E1 -5497.728,E2 -5497.728} C_VEL
LIN {X 0,Y 509.776,Z 447.034,A -85,B 0,C 180,E1 -5498.524,E2 -5498.524} C_VEL
LIN {X 0,Y 509.994,Z 439.108,A -85,B 0,C 180,E1 -5499.219,E2 -5499.219} C_VEL
LIN {X 0,Y 510.172,Z 430.736,A -85,B 0,C 180,E1 -5499.816,E2 -5499.816} C_VEL
LIN {X 0,Y 510.427,Z 420.052,A -85,B 0,C 180,E1 -5500.412,E2 -5500.412} C_VEL
LIN {X 0,Y 510.433,Z 410.079,A -85,B 0,C 180,E1 -5500.814,E2 -5500.814} C_VEL
LIN {X 0,Y 509.338,Z 399.903,A -85,B 0,C 180,E1 -5501.139,E2 -5501.139} C_VEL
LIN {X 0,Y 509.437,Z 389.603,A -85,B 0,C 180,E1 -5504.379,E2 -5504.379} C_VEL
LIN {X 0,Y 509.536,Z 380.5,A -85,B 0,C 180,E1 -5507.251,E2 -5507.251} C_VEL
LIN {X 0,Y 509.698,Z 372.855,A -85,B 0,C 180,E1 -5509.745,E2 -5509.745} C_VEL
LIN {X 0,Y 509.864,Z 362.616,A -85,B 0,C 180,E1 -5513.133,E2 -5513.133} C_VEL
LIN {X 0,Y 510.081,Z 353.732,A -85,B 0,C 180,E1 -5516.162,E2 -5516.162} C_VEL
LIN {X 0,Y 510.412,Z 345.039,A -85,B 0,C 180,E1 -5519.263,E2 -5519.263} C_VEL
LIN {X 0,Y 510.695,Z 337.709,A -85,B 0,C 180,E1 -5521.994,E2 -5521.994} C_VEL
LIN {X 0,Y 510.573,Z 334.105,A -85,B 0,C 180,E1 -5523.409,E2 -5523.409} C_VEL
LIN {X 0,Y 509.845,Z 329.791,A -85,B 0,C 180,E1 -5525.257,E2 -5525.257} C_VEL
LIN {X 0,Y 509.855,Z 329.792,A -85,B 0,C 180,E1 -5528.338,E2 -5528.338} C_VEL
LIN {X 0,Y 509.861,Z 329.793,A -85,B 0,C 180,E1 -5531.426,E2 -5531.426} C_VEL
LIN {X 0,Y 509.845,Z 329.792,A -85,B 0,C 180,E1 -5534.67,E2 -5534.67} C_VEL
LIN {X 0,Y 509.839,Z 329.794,A -85,B 0,C 180,E1 -5537.51,E2 -5537.51} C_VEL
LIN {X 0,Y 509.844,Z 329.79,A -85,B 0,C 180,E1 -5540.647,E2 -5540.647} C_VEL
LIN {X 0,Y 509.831,Z 329.794,A -85,B 0,C 180,E1 -5543.647,E2 -5543.647} C_VEL
LIN {X 0,Y 509.848,Z 329.79,A -85,B 0,C 180,E1 -5546.538,E2 -5546.538} C_VEL
LIN {X 0,Y 509.849,Z 329.792,A -85,B 0,C 180,E1 -5549.334,E2 -5549.334} C_VEL
LIN {X 0,Y 509.891,Z 329.785,A -85,B 0,C 180,E1 -5552.054,E2 -5552.054} C_VEL
LIN {X 0,Y 509.882,Z 329.785,A -85,B 0,C 180,E1 -5554.704,E2 -5554.704} C_VEL
LIN {X 0,Y 509.833,Z 329.793,A -85,B 0,C 180,E1 -5557.458,E2 -5557.458} C_VEL
LIN {X 0,Y 509.922,Z 329.782,A -85,B 0,C 180,E1 -5559.844,E2 -5559.844} C_VEL
LIN {X 0,Y 509.878,Z 329.786,A -85,B 0,C 180,E1 -5563.174,E2 -5563.174} C_VEL
LIN {X 0,Y 509.868,Z 329.788,A -85,B 0,C 180,E1 -5565.634,E2 -5565.634} C_VEL
LIN {X 0,Y 509.918,Z 329.781,A -85,B 0,C 180,E1 -5568.874,E2 -5568.874} C_VEL
LIN {X 0,Y 509.927,Z 329.781,A -85,B 0,C 180,E1 -5572.077,E2 -5572.077} C_VEL
LIN {X 0,Y 509.98,Z 329.774,A -85,B 0,C 180,E1 -5574.464,E2 -5574.464} C_VEL
LIN {X 0,Y 510.054,Z 329.767,A -85,B 0,C 180,E1 -5577.63,E2 -5577.63} C_VEL
LIN {X 0,Y 510.069,Z 329.762,A -85,B 0,C 180,E1 -5580.789,E2 -5580.789} C_VEL
LIN {X 0,Y 509.956,Z 329.776,A -85,B 0,C 180,E1 -5583.159,E2 -5583.159} C_VEL
LIN {X 0,Y 509.964,Z 329.776,A -85,B 0,C 180,E1 -5586.329,E2 -5586.329} C_VEL
LIN {X 0,Y 509.885,Z 329.788,A -85,B 0,C 180,E1 -5589.52,E2 -5589.52} C_VEL
LIN {X 0,Y 509.908,Z 329.785,A -85,B 0,C 180,E1 -5591.931,E2 -5591.931} C_VEL
LIN {X 0,Y 509.897,Z 329.787,A -85,B 0,C 180,E1 -5595.241,E2 -5595.241} C_VEL
LIN {X 0,Y 509.785,Z 329.801,A -85,B 0,C 180,E1 -5597.963,E2 -5597.963} C_VEL
LIN {X 0,Y 509.576,Z 329.93,A -85,B 0,C 180,E1 -5599.329,E2 -5599.329} C_VEL
LIN {X 0,Y 509.492,Z 334.023,A -85,B 0,C 180,E1 -5602.449,E2 -5602.449} C_VEL
LIN {X 0,Y 509.449,Z 337.802,A -85,B 0,C 180,E1 -5605.318,E2 -5605.318} C_VEL
LIN {X 0,Y 509.363,Z 341.353,A -85,B 0,C 180,E1 -5607.987,E2 -5607.987} C_VEL
LIN {X 0,Y 509.306,Z 344.978,A -85,B 0,C 180,E1 -5610.7,E2 -5610.7} C_VEL
LIN {X 0,Y 509.244,Z 348.814,A -85,B 0,C 180,E1 -5613.505,E2 -5613.505} C_VEL
LIN {X 0,Y 509.176,Z 352.759,A -85,B 0,C 180,E1 -5616.405,E2 -5616.405} C_VEL
LIN {X 0,Y 509.189,Z 356.356,A -85,B 0,C 180,E1 -5618.997,E2 -5618.997} C_VEL
LIN {X 0,Y 510.65,Z 366.193,A -85,B 0,C 180,E1 -5619.348,E2 -5619.348} C_VEL
LIN {X 0,Y 510.504,Z 375.251,A -85,B 0,C 180,E1 -5619.751,E2 -5619.751} C_VEL
LIN {X 0,Y 510.331,Z 384.104,A -85,B 0,C 180,E1 -5620.262,E2 -5620.262} C_VEL
LIN {X 0,Y 510.09,Z 392.363,A -85,B 0,C 180,E1 -5620.862,E2 -5620.862} C_VEL
LIN {X 0,Y 509.946,Z 399.86,A -85,B 0,C 180,E1 -5621.531,E2 -5621.531} C_VEL
LIN {X 0,Y 509.791,Z 405.773,A -85,B 0,C 180,E1 -5622.162,E2 -5622.162} C_VEL
LIN {X 0,Y 509.676,Z 410.674,A -85,B 0,C 180,E1 -5622.769,E2 -5622.769} C_VEL
LIN {X 0,Y 509.528,Z 416.303,A -85,B 0,C 180,E1 -5623.601,E2 -5623.601} C_VEL
LIN {X 0,Y 509.414,Z 420.848,A -85,B 0,C 180,E1 -5624.409,E2 -5624.409} C_VEL
LIN {X 0,Y 509.358,Z 424.845,A -85,B 0,C 180,E1 -5625.276,E2 -5625.276} C_VEL
LIN {X 0,Y 509.248,Z 428.709,A -85,B 0,C 180,E1 -5626.366,E2 -5626.366} C_VEL
LIN {X 0,Y 509.192,Z 431.048,A -85,B 0,C 180,E1 -5627.248,E2 -5627.248} C_VEL
LIN {X 0,Y 508.476,Z 432.407,A -85,B 0,C 180,E1 -5627.893,E2 -5627.893} C_VEL
LIN {X 0,Y 505.546,Z 433.919,A -85,B 0,C 180,E1 -5628.951,E2 -5628.951} C_VEL
LIN {X 0,Y 502.647,Z 434.522,A -85,B 0,C 180,E1 -5630.029,E2 -5630.029} C_VEL
LIN {X 0,Y 501.99,Z 434.315,A -85,B 0,C 180,E1 -5630.701,E2 -5630.701} C_VEL
LIN {X 0,Y 502.009,Z 433.086,A -85,B 0,C 180,E1 -5631.975,E2 -5631.975} C_VEL
LIN {X 0,Y 502.077,Z 431.142,A -85,B 0,C 180,E1 -5632.993,E2 -5632.993} C_VEL
LIN {X 0,Y 502.202,Z 427.468,A -85,B 0,C 180,E1 -5634.258,E2 -5634.258} C_VEL
LIN {X 0,Y 502.268,Z 423.1,A -85,B 0,C 180,E1 -5635.341,E2 -5635.341} C_VEL
LIN {X 0,Y 502.396,Z 418.673,A -85,B 0,C 180,E1 -5636.215,E2 -5636.215} C_VEL
LIN {X 0,Y 502.54,Z 413.584,A -85,B 0,C 180,E1 -5637.042,E2 -5637.042} C_VEL
LIN {X 0,Y 502.735,Z 407.063,A -85,B 0,C 180,E1 -5637.911,E2 -5637.911} C_VEL
LIN {X 0,Y 502.952,Z 400.05,A -85,B 0,C 180,E1 -5638.679,E2 -5638.679} C_VEL
LIN {X 0,Y 503.082,Z 392.738,A -85,B 0,C 180,E1 -5639.342,E2 -5639.342} C_VEL
LIN {X 0,Y 503.322,Z 384.322,A -85,B 0,C 180,E1 -5639.962,E2 -5639.962} C_VEL
LIN {X 0,Y 503.522,Z 374.631,A -85,B 0,C 180,E1 -5640.526,E2 -5640.526} C_VEL
LIN {X 0,Y 503.585,Z 365.444,A -85,B 0,C 180,E1 -5640.932,E2 -5640.932} C_VEL
LIN {X 0,Y 502.134,Z 356.454,A -85,B 0,C 180,E1 -5641.269,E2 -5641.269} C_VEL
LIN {X 0,Y 502.156,Z 352.232,A -85,B 0,C 180,E1 -5644.286,E2 -5644.286} C_VEL
LIN {X 0,Y 502.174,Z 348.595,A -85,B 0,C 180,E1 -5646.929,E2 -5646.929} C_VEL
LIN {X 0,Y 502.221,Z 343.899,A -85,B 0,C 180,E1 -5650.375,E2 -5650.375} C_VEL
LIN {X 0,Y 502.291,Z 340.466,A -85,B 0,C 180,E1 -5652.912,E2 -5652.912} C_VEL
LIN {X 0,Y 502.32,Z 337.118,A -85,B 0,C 180,E1 -5655.413,E2 -5655.413} C_VEL
LIN {X 0,Y 502.487,Z 332.724,A -85,B 0,C 180,E1 -5658.707,E2 -5658.707} C_VEL
LIN {X 0,Y 502.495,Z 330.708,A -85,B 0,C 180,E1 -5660.337,E2 -5660.337} C_VEL
LIN {X 0,Y 502.905,Z 330.654,A -85,B 0,C 180,E1 -5662.833,E2 -5662.833} C_VEL
LIN {X 0,Y 502.864,Z 330.659,A -85,B 0,C 180,E1 -5665.189,E2 -5665.189} C_VEL
LIN {X 0,Y 503.014,Z 330.641,A -85,B 0,C 180,E1 -5667.597,E2 -5667.597} C_VEL
LIN {X 0,Y 503.015,Z 330.642,A -85,B 0,C 180,E1 -5669.999,E2 -5669.999} C_VEL
LIN {X 0,Y 503.017,Z 330.641,A -85,B 0,C 180,E1 -5672.401,E2 -5672.401} C_VEL
LIN {X 0,Y 502.949,Z 330.65,A -85,B 0,C 180,E1 -5675.612,E2 -5675.612} C_VEL
LIN {X 0,Y 502.891,Z 330.659,A -85,B 0,C 180,E1 -5678.032,E2 -5678.032} C_VEL
LIN {X 0,Y 502.883,Z 330.657,A -85,B 0,C 180,E1 -5681.282,E2 -5681.282} C_VEL
LIN {X 0,Y 502.832,Z 330.662,A -85,B 0,C 180,E1 -5684.57,E2 -5684.57} C_VEL
LIN {X 0,Y 502.849,Z 330.663,A -85,B 0,C 180,E1 -5687.906,E2 -5687.906} C_VEL
LIN {X 0,Y 502.815,Z 330.666,A -85,B 0,C 180,E1 -5690.536,E2 -5690.536} C_VEL
LIN {X 0,Y 502.783,Z 330.671,A -85,B 0,C 180,E1 -5693.04,E2 -5693.04} C_VEL
LIN {X 0,Y 502.827,Z 330.665,A -85,B 0,C 180,E1 -5695.675,E2 -5695.675} C_VEL
LIN {X 0,Y 502.828,Z 330.664,A -85,B 0,C 180,E1 -5698.372,E2 -5698.372} C_VEL
LIN {X 0,Y 502.783,Z 330.671,A -85,B 0,C 180,E1 -5701.499,E2 -5701.499} C_VEL
LIN {X 0,Y 502.793,Z 330.668,A -85,B 0,C 180,E1 -5704.445,E2 -5704.445} C_VEL
LIN {X 0,Y 502.769,Z 330.674,A -85,B 0,C 180,E1 -5707.179,E2 -5707.179} C_VEL
LIN {X 0,Y 502.812,Z 330.665,A -85,B 0,C 180,E1 -5710.011,E2 -5710.011} C_VEL
LIN {X 0,Y 502.812,Z 330.667,A -85,B 0,C 180,E1 -5712.202,E2 -5712.202} C_VEL
LIN {X 0,Y 502.785,Z 330.671,A -85,B 0,C 180,E1 -5715.468,E2 -5715.468} C_VEL
LIN {X 0,Y 502.814,Z 330.666,A -85,B 0,C 180,E1 -5717.864,E2 -5717.864} C_VEL
LIN {X 0,Y 502.807,Z 330.667,A -85,B 0,C 180,E1 -5721.026,E2 -5721.026} C_VEL
LIN {X 0,Y 502.772,Z 330.672,A -85,B 0,C 180,E1 -5724.167,E2 -5724.167} C_VEL
LIN {X 0,Y 502.818,Z 330.666,A -85,B 0,C 180,E1 -5726.993,E2 -5726.993} C_VEL
LIN {X 0,Y 502.816,Z 330.665,A -85,B 0,C 180,E1 -5730.062,E2 -5730.062} C_VEL
LIN {X 0,Y 502.82,Z 330.666,A -85,B 0,C 180,E1 -5732.534,E2 -5732.534} C_VEL
LIN {X 0,Y 502.823,Z 330.665,A -85,B 0,C 180,E1 -5735.297,E2 -5735.297} C_VEL
LIN {X 0,Y 502.797,Z 330.67,A -85,B 0,C 180,E1 -5737.828,E2 -5737.828} C_VEL
LIN {X 0,Y 502.813,Z 330.667,A -85,B 0,C 180,E1 -5740.401,E2 -5740.401} C_VEL
LIN {X 0,Y 502.823,Z 330.664,A -85,B 0,C 180,E1 -5742.932,E2 -5742.932} C_VEL
LIN {X 0,Y 502.832,Z 330.663,A -85,B 0,C 180,E1 -5745.43,E2 -5745.43} C_VEL
LIN {X 0,Y 502.88,Z 330.658,A -85,B 0,C 180,E1 -5748.718,E2 -5748.718} C_VEL
LIN {X 0,Y 502.89,Z 330.658,A -85,B 0,C 180,E1 -5751.967,E2 -5751.967} C_VEL
LIN {X 0,Y 502.929,Z 330.653,A -85,B 0,C 180,E1 -5754.387,E2 -5754.387} C_VEL
LIN {X 0,Y 503.016,Z 330.641,A -85,B 0,C 180,E1 -5757.599,E2 -5757.599} C_VEL
LIN {X 0,Y 503.026,Z 330.64,A -85,B 0,C 180,E1 -5760.801,E2 -5760.801} C_VEL
LIN {X 0,Y 502.894,Z 330.657,A -85,B 0,C 180,E1 -5763.205,E2 -5763.205} C_VEL
LIN {X 0,Y 502.917,Z 330.654,A -85,B 0,C 180,E1 -5766.42,E2 -5766.42} C_VEL
LIN {X 0,Y 502.865,Z 330.659,A -85,B 0,C 180,E1 -5768.844,E2 -5768.844} C_VEL
LIN {X 0,Y 502.883,Z 330.657,A -85,B 0,C 180,E1 -5772.101,E2 -5772.101} C_VEL
LIN {X 0,Y 502.838,Z 330.665,A -85,B 0,C 180,E1 -5775.401,E2 -5775.401} C_VEL
LIN {X 0,Y 502.837,Z 330.662,A -85,B 0,C 180,E1 -5778.123,E2 -5778.123} C_VEL
LIN {X 0,Y 502.819,Z 330.665,A -85,B 0,C 180,E1 -5780.537,E2 -5780.537} C_VEL
LIN {X 0,Y 502.788,Z 330.669,A -85,B 0,C 180,E1 -5783.041,E2 -5783.041} C_VEL
LIN {X 0,Y 502.833,Z 330.664,A -85,B 0,C 180,E1 -5785.676,E2 -5785.676} C_VEL
LIN {X 0,Y 502.835,Z 330.664,A -85,B 0,C 180,E1 -5788.374,E2 -5788.374} C_VEL
LIN {X 0,Y 502.786,Z 330.669,A -85,B 0,C 180,E1 -5791.5,E2 -5791.5} C_VEL
LIN {X 0,Y 502.8,Z 330.667,A -85,B 0,C 180,E1 -5794.446,E2 -5794.446} C_VEL
LIN {X 0,Y 502.774,Z 330.673,A -85,B 0,C 180,E1 -5797.18,E2 -5797.18} C_VEL
LIN {X 0,Y 502.781,Z 330.669,A -85,B 0,C 180,E1 -5800.016,E2 -5800.016} C_VEL
LIN {X 0,Y 502.797,Z 330.669,A -85,B 0,C 180,E1 -5802.2,E2 -5802.2} C_VEL
LIN {X 0,Y 502.795,Z 330.67,A -85,B 0,C 180,E1 -5805.469,E2 -5805.469} C_VEL
LIN {X 0,Y 502.825,Z 330.665,A -85,B 0,C 180,E1 -5807.865,E2 -5807.865} C_VEL
LIN {X 0,Y 502.798,Z 330.667,A -85,B 0,C 180,E1 -5811.025,E2 -5811.025} C_VEL
LIN {X 0,Y 502.842,Z 330.663,A -85,B 0,C 180,E1 -5814.549,E2 -5814.549} C_VEL
LIN {X 0,Y 502.909,Z 330.988,A -85,B 0,C 180,E1 -5814.8,E2 -5814.8} C_VEL
LIN {X 0,Y 503.741,Z 336.544,A -85,B 0,C 180,E1 -5817.037,E2 -5817.037} C_VEL
LIN {X 0,Y 503.632,Z 341.506,A -85,B 0,C 180,E1 -5818.916,E2 -5818.916} C_VEL
LIN {X 0,Y 503.262,Z 350.237,A -85,B 0,C 180,E1 -5822.108,E2 -5822.108} C_VEL
LIN {X 0,Y 502.992,Z 359.025,A -85,B 0,C 180,E1 -5825.219,E2 -5825.219} C_VEL
LIN {X 0,Y 502.781,Z 366.608,A -85,B 0,C 180,E1 -5827.828,E2 -5827.828} C_VEL
LIN {X 0,Y 502.603,Z 375.482,A -85,B 0,C 180,E1 -5830.817,E2 -5830.817} C_VEL
LIN {X 0,Y 502.463,Z 385.765,A -85,B 0,C 180,E1 -5834.173,E2 -5834.173} C_VEL
LIN {X 0,Y 502.3,Z 395.97,A -85,B 0,C 180,E1 -5837.476,E2 -5837.476} C_VEL
LIN {X 0,Y 502.263,Z 399.86,A -85,B 0,C 180,E1 -5838.73,E2 -5838.73} C_VEL
LIN {X 0,Y 503.508,Z 411.454,A -85,B 0,C 180,E1 -5839.089,E2 -5839.089} C_VEL
LIN {X 0,Y 503.371,Z 421.797,A -85,B 0,C 180,E1 -5839.544,E2 -5839.544} C_VEL
LIN {X 0,Y 503.155,Z 430.539,A -85,B 0,C 180,E1 -5840.047,E2 -5840.047} C_VEL
LIN {X 0,Y 502.978,Z 438.892,A -85,B 0,C 180,E1 -5840.653,E2 -5840.653} C_VEL
LIN {X 0,Y 502.727,Z 446.796,A -85,B 0,C 180,E1 -5841.358,E2 -5841.358} C_VEL
LIN {X 0,Y 502.559,Z 454.192,A -85,B 0,C 180,E1 -5842.165,E2 -5842.165} C_VEL
LIN {X 0,Y 502.365,Z 461.7,A -85,B 0,C 180,E1 -5843.172,E2 -5843.172} C_VEL
LIN {X 0,Y 502.267,Z 468.561,A -85,B 0,C 180,E1 -5844.38,E2 -5844.38} C_VEL
LIN {X 0,Y 502.136,Z 473.763,A -85,B 0,C 180,E1 -5845.586,E2 -5845.586} C_VEL
LIN {X 0,Y 502.166,Z 476.428,A -85,B 0,C 180,E1 -5846.39,E2 -5846.39} C_VEL
LIN {X 0,Y 502.123,Z 479.344,A -85,B 0,C 180,E1 -5847.595,E2 -5847.595} C_VEL
LIN {X 0,Y 502.035,Z 480.6,A -85,B 0,C 180,E1 -5848.397,E2 -5848.397} C_VEL
LIN {X 0,Y 501.988,Z 481.379,A -85,B 0,C 180,E1 -5849.199,E2 -5849.199} C_VEL
LIN {X 0,Y 501.982,Z 481.67,A -85,B 0,C 180,E1 -5850.001,E2 -5850.001} C_VEL
LIN {X 0,Y 501.988,Z 481.369,A -85,B 0,C 180,E1 -5850.803,E2 -5850.803} C_VEL
LIN {X 0,Y 502.035,Z 480.581,A -85,B 0,C 180,E1 -5851.605,E2 -5851.605} C_VEL
LIN {X 0,Y 502.123,Z 479.316,A -85,B 0,C 180,E1 -5852.408,E2 -5852.408} C_VEL
LIN {X 0,Y 502.164,Z 476.384,A -85,B 0,C 180,E1 -5853.612,E2 -5853.612} C_VEL
LIN {X 0,Y 502.135,Z 473.709,A -85,B 0,C 180,E1 -5854.416,E2 -5854.416} C_VEL
LIN {X 0,Y 502.268,Z 468.485,A -85,B 0,C 180,E1 -5855.622,E2 -5855.622} C_VEL
LIN {X 0,Y 502.405,Z 461.601,A -85,B 0,C 180,E1 -5856.829,E2 -5856.829} C_VEL
LIN {X 0,Y 502.561,Z 454.08,A -85,B 0,C 180,E1 -5857.838,E2 -5857.838} C_VEL
LIN {X 0,Y 502.715,Z 446.666,A -85,B 0,C 180,E1 -5858.644,E2 -5858.644} C_VEL
LIN {X 0,Y 502.978,Z 438.738,A -85,B 0,C 180,E1 -5859.349,E2 -5859.349} C_VEL
LIN {X 0,Y 503.154,Z 430.361,A -85,B 0,C 180,E1 -5859.955,E2 -5859.955} C_VEL
LIN {X 0,Y 503.412,Z 419.669,A -85,B 0,C 180,E1 -5860.559,E2 -5860.559} C_VEL
LIN {X 0,Y 503.5,Z 411.227,A -85,B 0,C 180,E1 -5860.913,E2 -5860.913} C_VEL
LIN {X 0,Y 502.255,Z 399.546,A -85,B 0,C 180,E1 -5861.298,E2 -5861.298} C_VEL
LIN {X 0,Y 502.374,Z 389.242,A -85,B 0,C 180,E1 -5864.586,E2 -5864.586} C_VEL
LIN {X 0,Y 502.481,Z 380.231,A -85,B 0,C 180,E1 -5867.501,E2 -5867.501} C_VEL
LIN {X 0,Y 502.675,Z 371.311,A -85,B 0,C 180,E1 -5870.459,E2 -5870.459} C_VEL
LIN {X 0,Y 502.822,Z 362.343,A -85,B 0,C 180,E1 -5873.476,E2 -5873.476} C_VEL
LIN {X 0,Y 503.057,Z 354.833,A -85,B 0,C 180,E1 -5876.109,E2 -5876.109} C_VEL
LIN {X 0,Y 503.395,Z 346.167,A -85,B 0,C 180,E1 -5879.252,E2 -5879.252} C_VEL
LIN {X 0,Y 503.691,Z 338.856,A -85,B 0,C 180,E1 -5882.021,E2 -5882.021} C_VEL
LIN {X 0,Y 503.674,Z 336.007,A -85,B 0,C 180,E1 -5883.153,E2 -5883.153} C_VEL
LIN {X 0,Y 502.813,Z 330.667,A -85,B 0,C 180,E1 -5885.456,E2 -5885.456} C_VEL
LIN {X 0,Y 502.799,Z 330.67,A -85,B 0,C 180,E1 -5888.486,E2 -5888.486} C_VEL
LIN {X 0,Y 502.825,Z 330.668,A -85,B 0,C 180,E1 -5891.066,E2 -5891.066} C_VEL
LIN {X 0,Y 502.792,Z 330.671,A -85,B 0,C 180,E1 -5894.53,E2 -5894.53} C_VEL
LIN {X 0,Y 502.801,Z 330.669,A -85,B 0,C 180,E1 -5897.861,E2 -5897.861} C_VEL
LIN {X 0,Y 502.789,Z 330.67,A -85,B 0,C 180,E1 -5900.246,E2 -5900.246} C_VEL
LIN {X 0,Y 502.779,Z 330.671,A -85,B 0,C 180,E1 -5903.053,E2 -5903.053} C_VEL
LIN {X 0,Y 502.796,Z 330.67,A -85,B 0,C 180,E1 -5906.005,E2 -5906.005} C_VEL
LIN {X 0,Y 502.801,Z 330.668,A -85,B 0,C 180,E1 -5908.857,E2 -5908.857} C_VEL
LIN {X 0,Y 502.847,Z 330.664,A -85,B 0,C 180,E1 -5911.706,E2 -5911.706} C_VEL
LIN {X 0,Y 502.846,Z 330.663,A -85,B 0,C 180,E1 -5914.324,E2 -5914.324} C_VEL
LIN {X 0,Y 502.81,Z 330.667,A -85,B 0,C 180,E1 -5917.297,E2 -5917.297} C_VEL
LIN {X 0,Y 502.829,Z 330.664,A -85,B 0,C 180,E1 -5920.4,E2 -5920.4} C_VEL
LIN {X 0,Y 502.824,Z 330.664,A -85,B 0,C 180,E1 -5922.931,E2 -5922.931} C_VEL
LIN {X 0,Y 502.85,Z 330.662,A -85,B 0,C 180,E1 -5925.429,E2 -5925.429} C_VEL
LIN {X 0,Y 502.883,Z 330.657,A -85,B 0,C 180,E1 -5928.716,E2 -5928.716} C_VEL
LIN {X 0,Y 502.886,Z 330.658,A -85,B 0,C 180,E1 -5931.966,E2 -5931.966} C_VEL
LIN {X 0,Y 502.933,Z 330.652,A -85,B 0,C 180,E1 -5934.386,E2 -5934.386} C_VEL
LIN {X 0,Y 503.023,Z 330.642,A -85,B 0,C 180,E1 -5937.597,E2 -5937.597} C_VEL
LIN {X 0,Y 503.032,Z 330.641,A -85,B 0,C 180,E1 -5939.999,E2 -5939.999} C_VEL
LIN {X 0,Y 503.025,Z 330.643,A -85,B 0,C 180,E1 -5942.401,E2 -5942.401} C_VEL
LIN {X 0,Y 502.939,Z 330.65,A -85,B 0,C 180,E1 -5945.613,E2 -5945.613} C_VEL
LIN {X 0,Y 502.884,Z 330.658,A -85,B 0,C 180,E1 -5948.033,E2 -5948.033} C_VEL
LIN {X 0,Y 502.881,Z 330.658,A -85,B 0,C 180,E1 -5951.282,E2 -5951.282} C_VEL
LIN {X 0,Y 502.848,Z 330.664,A -85,B 0,C 180,E1 -5954.57,E2 -5954.57} C_VEL
LIN {X 0,Y 502.802,Z 330.669,A -85,B 0,C 180,E1 -5957.068,E2 -5957.068} C_VEL
LIN {X 0,Y 502.614,Z 330.694,A -85,B 0,C 180,E1 -5958.759,E2 -5958.759} C_VEL
LIN {X 0,Y 502.511,Z 331.086,A -85,B 0,C 180,E1 -5959.611,E2 -5959.611} C_VEL
LIN {X 0,Y 502.439,Z 334.949,A -85,B 0,C 180,E1 -5962.601,E2 -5962.601} C_VEL
LIN {X 0,Y 502.35,Z 338.997,A -85,B 0,C 180,E1 -5965.701,E2 -5965.701} C_VEL
LIN {X 0,Y 502.288,Z 342.585,A -85,B 0,C 180,E1 -5968.405,E2 -5968.405} C_VEL
LIN {X 0,Y 502.21,Z 346.57,A -85,B 0,C 180,E1 -5971.389,E2 -5971.389} C_VEL
LIN {X 0,Y 502.146,Z 350.538,A -85,B 0,C 180,E1 -5974.333,E2 -5974.333} C_VEL
LIN {X 0,Y 502.101,Z 354.292,A -85,B 0,C 180,E1 -5977.075,E2 -5977.075} C_VEL
LIN {X 0,Y 502.099,Z 356.733,A -85,B 0,C 180,E1 -5978.841,E2 -5978.841} C_VEL
LIN {X 0,Y 503.669,Z 366.862,A -85,B 0,C 180,E1 -5979.213,E2 -5979.213} C_VEL
LIN {X 0,Y 503.528,Z 375.649,A -85,B 0,C 180,E1 -5979.611,E2 -5979.611} C_VEL
LIN {X 0,Y 503.355,Z 383.9,A -85,B 0,C 180,E1 -5980.09,E2 -5980.09} C_VEL
LIN {X 0,Y 503.142,Z 391.427,A -85,B 0,C 180,E1 -5980.63,E2 -5980.63} C_VEL
LIN {X 0,Y 502.949,Z 399.236,A -85,B 0,C 180,E1 -5981.317,E2 -5981.317} C_VEL
LIN {X 0,Y 502.767,Z 405.717,A -85,B 0,C 180,E1 -5982.006,E2 -5982.006} C_VEL
LIN {X 0,Y 502.635,Z 411.209,A -85,B 0,C 180,E1 -5982.696,E2 -5982.696} C_VEL
LIN {X 0,Y 502.454,Z 417.269,A -85,B 0,C 180,E1 -5983.62,E2 -5983.62} C_VEL
LIN {X 0,Y 502.356,Z 421.886,A -85,B 0,C 180,E1 -5984.479,E2 -5984.479} C_VEL
LIN {X 0,Y 502.297,Z 424.502,A -85,B 0,C 180,E1 -5985.038,E2 -5985.038} C_VEL
LIN {X 0,Y 502.176,Z 428.579,A -85,B 0,C 180,E1 -5986.15,E2 -5986.15} C_VEL
LIN {X 0,Y 502.119,Z 431.473,A -85,B 0,C 180,E1 -5987.246,E2 -5987.246} C_VEL
LIN {X 0,Y 502.082,Z 432.756,A -85,B 0,C 180,E1 -5987.89,E2 -5987.89} C_VEL
LIN {X 0,Y 502.034,Z 434.209,A -85,B 0,C 180,E1 -5989.106,E2 -5989.106} C_VEL
LIN {X 0,Y 501.99,Z 434.457,A -85,B 0,C 180,E1 -5990.353,E2 -5990.353} C_VEL
LIN {X 0,Y 501.99,Z 434.315,A -85,B 0,C 180,E1 -5990.701,E2 -5990.701} C_VEL
LIN {X 0,Y 501.355,Z 433.909,A -85,B 0,C 180,E1 -5991.37,E2 -5991.37} C_VEL
LIN {X 0,Y 498.571,Z 432.558,A -85,B 0,C 180,E1 -5992.45,E2 -5992.45} C_VEL
LIN {X 0,Y 496.212,Z 430.793,A -85,B 0,C 180,E1 -5993.304,E2 -5993.304} C_VEL
LIN {X 0,Y 495.199,Z 428.992,A -85,B 0,C 180,E1 -5993.948,E2 -5993.948} C_VEL
LIN {X 0,Y 495.117,Z 428.293,A -85,B 0,C 180,E1 -5994.162,E2 -5994.162} C_VEL
LIN {X 0,Y 495.213,Z 423.447,A -85,B 0,C 180,E1 -5995.411,E2 -5995.411} C_VEL
LIN {X 0,Y 495.357,Z 418.413,A -85,B 0,C 180,E1 -5996.404,E2 -5996.404} C_VEL
LIN {X 0,Y 495.54,Z 412.195,A -85,B 0,C 180,E1 -5997.388,E2 -5997.388} C_VEL
LIN {X 0,Y 495.798,Z 404.52,A -85,B 0,C 180,E1 -5998.366,E2 -5998.366} C_VEL
LIN {X 0,Y 496.045,Z 394.741,A -85,B 0,C 180,E1 -5999.332,E2 -5999.332} C_VEL
LIN {X 0,Y 496.242,Z 387.194,A -85,B 0,C 180,E1 -5999.928,E2 -5999.928} C_VEL
LIN {X 0,Y 496.448,Z 378.622,A -85,B 0,C 180,E1 -6000.473,E2 -6000.473} C_VEL
LIN {X 0,Y 496.667,Z 370.182,A -85,B 0,C 180,E1 -6000.894,E2 -6000.894} C_VEL
LIN {X 0,Y 496.476,Z 365.127,A -85,B 0,C 180,E1 -6001.113,E2 -6001.113} C_VEL
LIN {X 0,Y 495.065,Z 356.744,A -85,B 0,C 180,E1 -6001.437,E2 -6001.437} C_VEL
LIN {X 0,Y 495.093,Z 353.336,A -85,B 0,C 180,E1 -6003.892,E2 -6003.892} C_VEL
LIN {X 0,Y 495.099,Z 349.657,A -85,B 0,C 180,E1 -6006.579,E2 -6006.579} C_VEL
LIN {X 0,Y 495.152,Z 344.896,A -85,B 0,C 180,E1 -6010.083,E2 -6010.083} C_VEL
LIN {X 0,Y 495.211,Z 341.444,A -85,B 0,C 180,E1 -6012.66,E2 -6012.66} C_VEL
LIN {X 0,Y 495.248,Z 338.067,A -85,B 0,C 180,E1 -6015.2,E2 -6015.2} C_VEL
LIN {X 0,Y 495.425,Z 333.656,A -85,B 0,C 180,E1 -6018.544,E2 -6018.544} C_VEL
LIN {X 0,Y 495.424,Z 331.589,A -85,B 0,C 180,E1 -6020.198,E2 -6020.198} C_VEL
LIN {X 0,Y 495.845,Z 331.534,A -85,B 0,C 180,E1 -6022.811,E2 -6022.811} C_VEL
LIN {X 0,Y 495.833,Z 331.535,A -85,B 0,C 180,E1 -6025.12,E2 -6025.12} C_VEL
LIN {X 0,Y 495.983,Z 331.517,A -85,B 0,C 180,E1 -6027.563,E2 -6027.563} C_VEL
LIN {X 0,Y 495.987,Z 331.517,A -85,B 0,C 180,E1 -6029.999,E2 -6029.999} C_VEL
LIN {X 0,Y 495.985,Z 331.517,A -85,B 0,C 180,E1 -6032.435,E2 -6032.435} C_VEL
LIN {X 0,Y 495.904,Z 331.529,A -85,B 0,C 180,E1 -6035.692,E2 -6035.692} C_VEL
LIN {X 0,Y 495.862,Z 331.534,A -85,B 0,C 180,E1 -6038.147,E2 -6038.147} C_VEL
LIN {X 0,Y 495.857,Z 331.533,A -85,B 0,C 180,E1 -6041.444,E2 -6041.444} C_VEL
LIN {X 0,Y 495.777,Z 331.541,A -85,B 0,C 180,E1 -6044.782,E2 -6044.782} C_VEL
LIN {X 0,Y 495.775,Z 331.543,A -85,B 0,C 180,E1 -6047.318,E2 -6047.318} C_VEL
LIN {X 0,Y 495.765,Z 331.545,A -85,B 0,C 180,E1 -6049.889,E2 -6049.889} C_VEL
LIN {X 0,Y 495.744,Z 331.548,A -85,B 0,C 180,E1 -6052.86,E2 -6052.86} C_VEL
LIN {X 0,Y 495.785,Z 331.543,A -85,B 0,C 180,E1 -6056.067,E2 -6056.067} C_VEL
LIN {X 0,Y 495.766,Z 331.545,A -85,B 0,C 180,E1 -6058.814,E2 -6058.814} C_VEL
LIN {X 0,Y 495.745,Z 331.546,A -85,B 0,C 180,E1 -6061.726,E2 -6061.726} C_VEL
LIN {X 0,Y 495.763,Z 331.544,A -85,B 0,C 180,E1 -6064.695,E2 -6064.695} C_VEL
LIN {X 0,Y 495.72,Z 331.55,A -85,B 0,C 180,E1 -6067.561,E2 -6067.561} C_VEL
LIN {X 0,Y 495.779,Z 331.541,A -85,B 0,C 180,E1 -6070.052,E2 -6070.052} C_VEL
LIN {X 0,Y 495.749,Z 331.546,A -85,B 0,C 180,E1 -6072.879,E2 -6072.879} C_VEL
LIN {X 0,Y 495.721,Z 331.55,A -85,B 0,C 180,E1 -6075.999,E2 -6075.999} C_VEL
LIN {X 0,Y 495.753,Z 331.546,A -85,B 0,C 180,E1 -6078.705,E2 -6078.705} C_VEL
LIN {X 0,Y 495.75,Z 331.546,A -85,B 0,C 180,E1 -6081.41,E2 -6081.41} C_VEL
LIN {X 0,Y 495.744,Z 331.548,A -85,B 0,C 180,E1 -6084.463,E2 -6084.463} C_VEL
LIN {X 0,Y 495.755,Z 331.545,A -85,B 0,C 180,E1 -6087.406,E2 -6087.406} C_VEL
LIN {X 0,Y 495.767,Z 331.545,A -85,B 0,C 180,E1 -6090.255,E2 -6090.255} C_VEL
LIN {X 0,Y 495.809,Z 331.538,A -85,B 0,C 180,E1 -6093.251,E2 -6093.251} C_VEL
LIN {X 0,Y 495.753,Z 331.544,A -85,B 0,C 180,E1 -6095.726,E2 -6095.726} C_VEL
LIN {X 0,Y 495.747,Z 331.547,A -85,B 0,C 180,E1 -6098.372,E2 -6098.372} C_VEL
LIN {X 0,Y 495.772,Z 331.544,A -85,B 0,C 180,E1 -6100.972,E2 -6100.972} C_VEL
LIN {X 0,Y 495.768,Z 331.544,A -85,B 0,C 180,E1 -6103.531,E2 -6103.531} C_VEL
LIN {X 0,Y 495.781,Z 331.544,A -85,B 0,C 180,E1 -6106.056,E2 -6106.056} C_VEL
LIN {X 0,Y 495.855,Z 331.534,A -85,B 0,C 180,E1 -6108.556,E2 -6108.556} C_VEL
LIN {X 0,Y 495.861,Z 331.532,A -85,B 0,C 180,E1 -6111.853,E2 -6111.853} C_VEL
LIN {X 0,Y 495.886,Z 331.53,A -85,B 0,C 180,E1 -6114.307,E2 -6114.307} C_VEL
LIN {X 0,Y 495.985,Z 331.517,A -85,B 0,C 180,E1 -6117.564,E2 -6117.564} C_VEL
LIN {X 0,Y 495.986,Z 331.517,A -85,B 0,C 180,E1 -6120.001,E2 -6120.001} C_VEL
LIN {X 0,Y 495.985,Z 331.516,A -85,B 0,C 180,E1 -6122.437,E2 -6122.437} C_VEL
LIN {X 0,Y 495.885,Z 331.531,A -85,B 0,C 180,E1 -6125.694,E2 -6125.694} C_VEL
LIN {X 0,Y 495.863,Z 331.532,A -85,B 0,C 180,E1 -6128.149,E2 -6128.149} C_VEL
LIN {X 0,Y 495.86,Z 331.533,A -85,B 0,C 180,E1 -6131.446,E2 -6131.446} C_VEL
LIN {X 0,Y 495.781,Z 331.54,A -85,B 0,C 180,E1 -6134.784,E2 -6134.784} C_VEL
LIN {X 0,Y 495.779,Z 331.543,A -85,B 0,C 180,E1 -6137.319,E2 -6137.319} C_VEL
LIN {X 0,Y 495.763,Z 331.546,A -85,B 0,C 180,E1 -6139.891,E2 -6139.891} C_VEL
LIN {X 0,Y 495.749,Z 331.547,A -85,B 0,C 180,E1 -6142.861,E2 -6142.861} C_VEL
LIN {X 0,Y 495.791,Z 331.542,A -85,B 0,C 180,E1 -6146.068,E2 -6146.068} C_VEL
LIN {X 0,Y 495.773,Z 331.545,A -85,B 0,C 180,E1 -6148.815,E2 -6148.815} C_VEL
LIN {X 0,Y 495.749,Z 331.546,A -85,B 0,C 180,E1 -6151.727,E2 -6151.727} C_VEL
LIN {X 0,Y 495.77,Z 331.545,A -85,B 0,C 180,E1 -6154.697,E2 -6154.697} C_VEL
LIN {X 0,Y 495.724,Z 331.549,A -85,B 0,C 180,E1 -6157.563,E2 -6157.563} C_VEL
LIN {X 0,Y 495.76,Z 331.546,A -85,B 0,C 180,E1 -6160.701,E2 -6160.701} C_VEL
LIN {X 0,Y 495.729,Z 331.547,A -85,B 0,C 180,E1 -6163.697,E2 -6163.697} C_VEL
LIN {X 0,Y 495.729,Z 331.548,A -85,B 0,C 180,E1 -6166.306,E2 -6166.306} C_VEL
LIN {X 0,Y 495.762,Z 331.546,A -85,B 0,C 180,E1 -6169.301,E2 -6169.301} C_VEL
LIN {X 0,Y 495.727,Z 331.548,A -85,B 0,C 180,E1 -6172.44,E2 -6172.44} C_VEL
LIN {X 0,Y 495.821,Z 331.654,A -85,B 0,C 180,E1 -6174.522,E2 -6174.522} C_VEL
LIN {X 0,Y 496.641,Z 336.71,A -85,B 0,C 180,E1 -6176.607,E2 -6176.607} C_VEL
LIN {X 0,Y 496.676,Z 341.41,A -85,B 0,C 180,E1 -6178.431,E2 -6178.431} C_VEL
LIN {X 0,Y 496.313,Z 349.319,A -85,B 0,C 180,E1 -6181.396,E2 -6181.396} C_VEL
LIN {X 0,Y 495.991,Z 357.599,A -85,B 0,C 180,E1 -6184.396,E2 -6184.396} C_VEL
LIN {X 0,Y 495.797,Z 365.358,A -85,B 0,C 180,E1 -6187.13,E2 -6187.13} C_VEL
LIN {X 0,Y 495.541,Z 375.292,A -85,B 0,C 180,E1 -6190.533,E2 -6190.533} C_VEL
LIN {X 0,Y 495.382,Z 385.435,A -85,B 0,C 180,E1 -6193.941,E2 -6193.941} C_VEL
LIN {X 0,Y 495.19,Z 394.372,A -85,B 0,C 180,E1 -6196.876,E2 -6196.876} C_VEL
LIN {X 0,Y 495.187,Z 399.538,A -85,B 0,C 180,E1 -6198.566,E2 -6198.566} C_VEL
LIN {X 0,Y 496.397,Z 411.095,A -85,B 0,C 180,E1 -6198.931,E2 -6198.931} C_VEL
LIN {X 0,Y 496.37,Z 421.449,A -85,B 0,C 180,E1 -6199.395,E2 -6199.395} C_VEL
LIN {X 0,Y 496.168,Z 430.194,A -85,B 0,C 180,E1 -6199.906,E2 -6199.906} C_VEL
LIN {X 0,Y 495.966,Z 438.548,A -85,B 0,C 180,E1 -6200.52,E2 -6200.52} C_VEL
LIN {X 0,Y 495.704,Z 446.454,A -85,B 0,C 180,E1 -6201.234,E2 -6201.234} C_VEL
LIN {X 0,Y 495.503,Z 453.852,A -85,B 0,C 180,E1 -6202.052,E2 -6202.052} C_VEL
LIN {X 0,Y 495.298,Z 461.363,A -85,B 0,C 180,E1 -6203.074,E2 -6203.074} C_VEL
LIN {X 0,Y 495.198,Z 468.228,A -85,B 0,C 180,E1 -6204.3,E2 -6204.3} C_VEL
LIN {X 0,Y 495.041,Z 473.429,A -85,B 0,C 180,E1 -6205.523,E2 -6205.523} C_VEL
LIN {X 0,Y 495.086,Z 476.096,A -85,B 0,C 180,E1 -6206.339,E2 -6206.339} C_VEL
LIN {X 0,Y 495.027,Z 479.012,A -85,B 0,C 180,E1 -6207.56,E2 -6207.56} C_VEL
LIN {X 0,Y 494.962,Z 480.269,A -85,B 0,C 180,E1 -6208.374,E2 -6208.374} C_VEL
LIN {X 0,Y 494.908,Z 481.048,A -85,B 0,C 180,E1 -6209.187,E2 -6209.187} C_VEL
LIN {X 0,Y 494.899,Z 481.338,A -85,B 0,C 180,E1 -6210.001,E2 -6210.001} C_VEL
LIN {X 0,Y 494.909,Z 481.035,A -85,B 0,C 180,E1 -6210.815,E2 -6210.815} C_VEL
LIN {X 0,Y 494.962,Z 480.245,A -85,B 0,C 180,E1 -6211.628,E2 -6211.628} C_VEL
LIN {X 0,Y 495.027,Z 478.979,A -85,B 0,C 180,E1 -6212.442,E2 -6212.442} C_VEL
LIN {X 0,Y 495.085,Z 476.042,A -85,B 0,C 180,E1 -6213.664,E2 -6213.664} C_VEL
LIN {X 0,Y 495.041,Z 473.364,A -85,B 0,C 180,E1 -6214.479,E2 -6214.479} C_VEL
LIN {X 0,Y 495.199,Z 468.136,A -85,B 0,C 180,E1 -6215.703,E2 -6215.703} C_VEL
LIN {X 0,Y 495.336,Z 461.245,A -85,B 0,C 180,E1 -6216.927,E2 -6216.927} C_VEL
LIN {X 0,Y 495.504,Z 453.718,A -85,B 0,C 180,E1 -6217.95,E2 -6217.95} C_VEL
LIN {X 0,Y 495.703,Z 446.301,A -85,B 0,C 180,E1 -6218.768,E2 -6218.768} C_VEL
LIN {X 0,Y 495.961,Z 438.367,A -85,B 0,C 180,E1 -6219.483,E2 -6219.483} C_VEL
LIN {X 0,Y 496.143,Z 429.986,A -85,B 0,C 180,E1 -6220.097,E2 -6220.097} C_VEL
LIN {X 0,Y 496.44,Z 419.287,A -85,B 0,C 180,E1 -6220.709,E2 -6220.709} C_VEL
LIN {X 0,Y 496.387,Z 410.833,A -85,B 0,C 180,E1 -6221.072,E2 -6221.072} C_VEL
LIN {X 0,Y 495.163,Z 399.188,A -85,B 0,C 180,E1 -6221.462,E2 -6221.462} C_VEL
LIN {X 0,Y 495.31,Z 388.946,A -85,B 0,C 180,E1 -6224.798,E2 -6224.798} C_VEL
LIN {X 0,Y 495.467,Z 378.86,A -85,B 0,C 180,E1 -6228.127,E2 -6228.127} C_VEL
LIN {X 0,Y 495.592,Z 371.034,A -85,B 0,C 180,E1 -6230.765,E2 -6230.765} C_VEL
LIN {X 0,Y 495.779,Z 362.159,A -85,B 0,C 180,E1 -6233.83,E2 -6233.83} C_VEL
LIN {X 0,Y 496.021,Z 354.9,A -85,B 0,C 180,E1 -6236.431,E2 -6236.431} C_VEL
LIN {X 0,Y 496.431,Z 346.068,A -85,B 0,C 180,E1 -6239.703,E2 -6239.703} C_VEL
LIN {X 0,Y 496.726,Z 338.803,A -85,B 0,C 180,E1 -6242.525,E2 -6242.525} C_VEL
LIN {X 0,Y 496.431,Z 335.25,A -85,B 0,C 180,E1 -6244.002,E2 -6244.002} C_VEL
LIN {X 0,Y 495.75,Z 331.548,A -85,B 0,C 180,E1 -6245.64,E2 -6245.64} C_VEL
LIN {X 0,Y 495.768,Z 331.545,A -85,B 0,C 180,E1 -6248.768,E2 -6248.768} C_VEL
LIN {X 0,Y 495.762,Z 331.551,A -85,B 0,C 180,E1 -6251.781,E2 -6251.781} C_VEL
LIN {X 0,Y 495.743,Z 331.551,A -85,B 0,C 180,E1 -6255.141,E2 -6255.141} C_VEL
LIN {X 0,Y 495.762,Z 331.545,A -85,B 0,C 180,E1 -6258.219,E2 -6258.219} C_VEL
LIN {X 0,Y 495.753,Z 331.547,A -85,B 0,C 180,E1 -6261.408,E2 -6261.408} C_VEL
LIN {X 0,Y 495.753,Z 331.547,A -85,B 0,C 180,E1 -6264.462,E2 -6264.462} C_VEL
LIN {X 0,Y 495.772,Z 331.544,A -85,B 0,C 180,E1 -6267.405,E2 -6267.405} C_VEL
LIN {X 0,Y 495.772,Z 331.544,A -85,B 0,C 180,E1 -6270.253,E2 -6270.253} C_VEL
LIN {X 0,Y 495.83,Z 331.537,A -85,B 0,C 180,E1 -6273.251,E2 -6273.251} C_VEL
LIN {X 0,Y 495.754,Z 331.546,A -85,B 0,C 180,E1 -6275.725,E2 -6275.725} C_VEL
LIN {X 0,Y 495.748,Z 331.546,A -85,B 0,C 180,E1 -6278.371,E2 -6278.371} C_VEL
LIN {X 0,Y 495.788,Z 331.542,A -85,B 0,C 180,E1 -6280.971,E2 -6280.971} C_VEL
LIN {X 0,Y 495.814,Z 331.538,A -85,B 0,C 180,E1 -6284.376,E2 -6284.376} C_VEL
LIN {X 0,Y 495.788,Z 331.542,A -85,B 0,C 180,E1 -6286.89,E2 -6286.89} C_VEL
LIN {X 0,Y 495.778,Z 331.545,A -85,B 0,C 180,E1 -6289.38,E2 -6289.38} C_VEL
LIN {X 0,Y 495.842,Z 331.537,A -85,B 0,C 180,E1 -6291.851,E2 -6291.851} C_VEL
LIN {X 0,Y 495.888,Z 331.531,A -85,B 0,C 180,E1 -6294.306,E2 -6294.306} C_VEL
LIN {X 0,Y 495.991,Z 331.518,A -85,B 0,C 180,E1 -6297.563,E2 -6297.563} C_VEL
LIN {X 0,Y 495.989,Z 331.516,A -85,B 0,C 180,E1 -6300.811,E2 -6300.811} C_VEL
LIN {X 0,Y 495.995,Z 331.518,A -85,B 0,C 180,E1 -6302.435,E2 -6302.435} C_VEL
LIN {X 0,Y 495.896,Z 331.528,A -85,B 0,C 180,E1 -6305.693,E2 -6305.693} C_VEL
LIN {X 0,Y 495.84,Z 331.536,A -85,B 0,C 180,E1 -6308.148,E2 -6308.148} C_VEL
LIN {X 0,Y 495.855,Z 331.533,A -85,B 0,C 180,E1 -6311.444,E2 -6311.444} C_VEL
LIN {X 0,Y 495.793,Z 331.542,A -85,B 0,C 180,E1 -6314.782,E2 -6314.782} C_VEL
LIN {X 0,Y 495.729,Z 331.551,A -85,B 0,C 180,E1 -6317.32,E2 -6317.32} C_VEL
LIN {X 0,Y 495.525,Z 331.577,A -85,B 0,C 180,E1 -6319.038,E2 -6319.038} C_VEL
LIN {X 0,Y 495.443,Z 333.109,A -85,B 0,C 180,E1 -6320.571,E2 -6320.571} C_VEL
LIN {X 0,Y 495.355,Z 336.764,A -85,B 0,C 180,E1 -6323.406,E2 -6323.406} C_VEL
LIN {X 0,Y 495.273,Z 340.229,A -85,B 0,C 180,E1 -6326.096,E2 -6326.096} C_VEL
LIN {X 0,Y 495.215,Z 343.809,A -85,B 0,C 180,E1 -6328.849,E2 -6328.849} C_VEL
LIN {X 0,Y 495.137,Z 347.611,A -85,B 0,C 180,E1 -6331.679,E2 -6331.679} C_VEL
LIN {X 0,Y 495.072,Z 351.494,A -85,B 0,C 180,E1 -6334.598,E2 -6334.598} C_VEL
LIN {X 0,Y 495.006,Z 355.64,A -85,B 0,C 180,E1 -6337.625,E2 -6337.625} C_VEL
LIN {X 0,Y 495.035,Z 357.049,A -85,B 0,C 180,E1 -6338.662,E2 -6338.662} C_VEL
LIN {X 0,Y 496.732,Z 367.73,A -85,B 0,C 180,E1 -6339.084,E2 -6339.084} C_VEL
LIN {X 0,Y 496.545,Z 376.552,A -85,B 0,C 180,E1 -6339.495,E2 -6339.495} C_VEL
LIN {X 0,Y 496.364,Z 385.2,A -85,B 0,C 180,E1 -6340.016,E2 -6340.016} C_VEL
LIN {X 0,Y 496.164,Z 391.923,A -85,B 0,C 180,E1 -6340.511,E2 -6340.511} C_VEL
LIN {X 0,Y 495.941,Z 399.36,A -85,B 0,C 180,E1 -6341.173,E2 -6341.173} C_VEL
LIN {X 0,Y 495.727,Z 406.581,A -85,B 0,C 180,E1 -6341.956,E2 -6341.956} C_VEL
LIN {X 0,Y 495.599,Z 412.031,A -85,B 0,C 180,E1 -6342.663,E2 -6342.663} C_VEL
LIN {X 0,Y 495.371,Z 418.298,A -85,B 0,C 180,E1 -6343.65,E2 -6343.65} C_VEL
LIN {X 0,Y 495.307,Z 422.343,A -85,B 0,C 180,E1 -6344.427,E2 -6344.427} C_VEL
LIN {X 0,Y 495.151,Z 427.089,A -85,B 0,C 180,E1 -6345.566,E2 -6345.566} C_VEL
LIN {X 0,Y 495.077,Z 429.719,A -85,B 0,C 180,E1 -6346.383,E2 -6346.383} C_VEL
LIN {X 0,Y 495.043,Z 431.485,A -85,B 0,C 180,E1 -6347.043,E2 -6347.043} C_VEL
LIN {X 0,Y 494.987,Z 433.502,A -85,B 0,C 180,E1 -6348.138,E2 -6348.138} C_VEL
LIN {X 0,Y 494.935,Z 434.593,A -85,B 0,C 180,E1 -6349.216,E2 -6349.216} C_VEL
LIN {X 0,Y 494.905,Z 434.82,A -85,B 0,C 180,E1 -6350.279,E2 -6350.279} C_VEL
LIN {X 0,Y 494.925,Z 434.189,A -85,B 0,C 180,E1 -6351.351,E2 -6351.351} C_VEL
LIN {X 0,Y 494.96,Z 432.2,A -85,B 0,C 180,E1 -6352.667,E2 -6352.667} C_VEL
LIN {X 0,Y 495.12,Z 428.826,A -85,B 0,C 180,E1 -6354.005,E2 -6354.005} C_VEL
LIN {X 0,Y 495.117,Z 428.293,A -85,B 0,C 180,E1 -6354.162,E2 -6354.162} C_VEL
LIN {X 0,Y 494.472,Z 426.119,A -85,B 0,C 180,E1 -6354.793,E2 -6354.793} C_VEL
LIN {X 0,Y 491.724,Z 422.028,A -85,B 0,C 180,E1 -6355.797,E2 -6355.797} C_VEL
LIN {X 0,Y 489.032,Z 417.212,A -85,B 0,C 180,E1 -6356.759,E2 -6356.759} C_VEL
LIN {X 0,Y 488.477,Z 413.719,A -85,B 0,C 180,E1 -6357.316,E2 -6357.316} C_VEL
LIN {X 0,Y 488.716,Z 407.2,A -85,B 0,C 180,E1 -6358.196,E2 -6358.196} C_VEL
LIN {X 0,Y 488.914,Z 401.569,A -85,B 0,C 180,E1 -6358.835,E2 -6358.835} C_VEL
LIN {X 0,Y 489.089,Z 393.938,A -85,B 0,C 180,E1 -6359.559,E2 -6359.559} C_VEL
LIN {X 0,Y 489.33,Z 385.928,A -85,B 0,C 180,E1 -6360.177,E2 -6360.177} C_VEL
LIN {X 0,Y 489.538,Z 378.144,A -85,B 0,C 180,E1 -6360.664,E2 -6360.664} C_VEL
LIN {X 0,Y 489.717,Z 369.494,A -85,B 0,C 180,E1 -6361.092,E2 -6361.092} C_VEL
LIN {X 0,Y 489.044,Z 363.049,A -85,B 0,C 180,E1 -6361.363,E2 -6361.363} C_VEL
LIN {X 0,Y 487.968,Z 357.051,A -85,B 0,C 180,E1 -6361.599,E2 -6361.599} C_VEL
LIN {X 0,Y 488.007,Z 353.201,A -85,B 0,C 180,E1 -6364.402,E2 -6364.402} C_VEL
LIN {X 0,Y 488.016,Z 349.431,A -85,B 0,C 180,E1 -6367.168,E2 -6367.168} C_VEL
LIN {X 0,Y 488.08,Z 345.926,A -85,B 0,C 180,E1 -6369.782,E2 -6369.782} C_VEL
LIN {X 0,Y 488.152,Z 342.417,A -85,B 0,C 180,E1 -6372.401,E2 -6372.401} C_VEL
LIN {X 0,Y 488.19,Z 339.024,A -85,B 0,C 180,E1 -6374.981,E2 -6374.981} C_VEL
LIN {X 0,Y 488.371,Z 334.565,A -85,B 0,C 180,E1 -6378.376,E2 -6378.376} C_VEL
LIN {X 0,Y 488.354,Z 332.47,A -85,B 0,C 180,E1 -6380.055,E2 -6380.055} C_VEL
LIN {X 0,Y 488.804,Z 332.411,A -85,B 0,C 180,E1 -6382.772,E2 -6382.772} C_VEL
LIN {X 0,Y 488.802,Z 332.411,A -85,B 0,C 180,E1 -6385.05,E2 -6385.05} C_VEL
LIN {X 0,Y 488.95,Z 332.394,A -85,B 0,C 180,E1 -6387.528,E2 -6387.528} C_VEL
LIN {X 0,Y 488.958,Z 332.393,A -85,B 0,C 180,E1 -6389.999,E2 -6389.999} C_VEL
LIN {X 0,Y 488.953,Z 332.392,A -85,B 0,C 180,E1 -6392.47,E2 -6392.47} C_VEL
LIN {X 0,Y 488.86,Z 332.407,A -85,B 0,C 180,E1 -6395.775,E2 -6395.775} C_VEL
LIN {X 0,Y 488.807,Z 332.411,A -85,B 0,C 180,E1 -6398.265,E2 -6398.265} C_VEL
LIN {X 0,Y 488.818,Z 332.41,A -85,B 0,C 180,E1 -6401.611,E2 -6401.611} C_VEL
LIN {X 0,Y 488.749,Z 332.416,A -85,B 0,C 180,E1 -6405,E2 -6405} C_VEL
LIN {X 0,Y 488.741,Z 332.418,A -85,B 0,C 180,E1 -6408.441,E2 -6408.441} C_VEL
LIN {X 0,Y 488.694,Z 332.424,A -85,B 0,C 180,E1 -6411.07,E2 -6411.07} C_VEL
LIN {X 0,Y 488.68,Z 332.429,A -85,B 0,C 180,E1 -6413.745,E2 -6413.745} C_VEL
LIN {X 0,Y 488.785,Z 332.413,A -85,B 0,C 180,E1 -6416.945,E2 -6416.945} C_VEL
LIN {X 0,Y 488.705,Z 332.423,A -85,B 0,C 180,E1 -6420.364,E2 -6420.364} C_VEL
LIN {X 0,Y 488.721,Z 332.424,A -85,B 0,C 180,E1 -6423.484,E2 -6423.484} C_VEL
LIN {X 0,Y 488.676,Z 332.427,A -85,B 0,C 180,E1 -6426.356,E2 -6426.356} C_VEL
LIN {X 0,Y 488.734,Z 332.421,A -85,B 0,C 180,E1 -6429.249,E2 -6429.249} C_VEL
LIN {X 0,Y 488.719,Z 332.422,A -85,B 0,C 180,E1 -6432.521,E2 -6432.521} C_VEL
LIN {X 0,Y 488.696,Z 332.425,A -85,B 0,C 180,E1 -6435.199,E2 -6435.199} C_VEL
LIN {X 0,Y 488.72,Z 332.421,A -85,B 0,C 180,E1 -6437.479,E2 -6437.479} C_VEL
LIN {X 0,Y 488.734,Z 332.422,A -85,B 0,C 180,E1 -6440.75,E2 -6440.75} C_VEL
LIN {X 0,Y 488.672,Z 332.427,A -85,B 0,C 180,E1 -6443.869,E2 -6443.869} C_VEL
LIN {X 0,Y 488.724,Z 332.422,A -85,B 0,C 180,E1 -6446.878,E2 -6446.878} C_VEL
LIN {X 0,Y 488.72,Z 332.42,A -85,B 0,C 180,E1 -6449.782,E2 -6449.782} C_VEL
LIN {X 0,Y 488.777,Z 332.414,A -85,B 0,C 180,E1 -6453.057,E2 -6453.057} C_VEL
LIN {X 0,Y 488.694,Z 332.426,A -85,B 0,C 180,E1 -6456.256,E2 -6456.256} C_VEL
LIN {X 0,Y 488.733,Z 332.419,A -85,B 0,C 180,E1 -6459.176,E2 -6459.176} C_VEL
LIN {X 0,Y 488.745,Z 332.419,A -85,B 0,C 180,E1 -6461.628,E2 -6461.628} C_VEL
LIN {X 0,Y 488.749,Z 332.418,A -85,B 0,C 180,E1 -6465,E2 -6465} C_VEL
LIN {X 0,Y 488.817,Z 332.412,A -85,B 0,C 180,E1 -6468.389,E2 -6468.389} C_VEL
LIN {X 0,Y 488.806,Z 332.411,A -85,B 0,C 180,E1 -6471.734,E2 -6471.734} C_VEL
LIN {X 0,Y 488.845,Z 332.407,A -85,B 0,C 180,E1 -6474.225,E2 -6474.225} C_VEL
LIN {X 0,Y 488.952,Z 332.393,A -85,B 0,C 180,E1 -6477.529,E2 -6477.529} C_VEL
LIN {X 0,Y 488.967,Z 332.391,A -85,B 0,C 180,E1 -6480.824,E2 -6480.824} C_VEL
LIN {X 0,Y 488.952,Z 332.392,A -85,B 0,C 180,E1 -6482.472,E2 -6482.472} C_VEL
LIN {X 0,Y 488.845,Z 332.407,A -85,B 0,C 180,E1 -6485.777,E2 -6485.777} C_VEL
LIN {X 0,Y 488.807,Z 332.41,A -85,B 0,C 180,E1 -6488.267,E2 -6488.267} C_VEL
LIN {X 0,Y 488.821,Z 332.412,A -85,B 0,C 180,E1 -6491.613,E2 -6491.613} C_VEL
LIN {X 0,Y 488.752,Z 332.417,A -85,B 0,C 180,E1 -6495.001,E2 -6495.001} C_VEL
LIN {X 0,Y 488.745,Z 332.418,A -85,B 0,C 180,E1 -6498.443,E2 -6498.443} C_VEL
LIN {X 0,Y 488.699,Z 332.424,A -85,B 0,C 180,E1 -6501.072,E2 -6501.072} C_VEL
LIN {X 0,Y 488.685,Z 332.427,A -85,B 0,C 180,E1 -6503.746,E2 -6503.746} C_VEL
LIN {X 0,Y 488.791,Z 332.413,A -85,B 0,C 180,E1 -6506.946,E2 -6506.946} C_VEL
LIN {X 0,Y 488.711,Z 332.422,A -85,B 0,C 180,E1 -6510.366,E2 -6510.366} C_VEL
LIN {X 0,Y 488.728,Z 332.422,A -85,B 0,C 180,E1 -6513.486,E2 -6513.486} C_VEL
LIN {X 0,Y 488.682,Z 332.426,A -85,B 0,C 180,E1 -6516.357,E2 -6516.357} C_VEL
LIN {X 0,Y 488.695,Z 332.426,A -85,B 0,C 180,E1 -6519.255,E2 -6519.255} C_VEL
LIN {X 0,Y 488.717,Z 332.423,A -85,B 0,C 180,E1 -6521.603,E2 -6521.603} C_VEL
LIN {X 0,Y 488.706,Z 332.424,A -85,B 0,C 180,E1 -6524.803,E2 -6524.803} C_VEL
LIN {X 0,Y 488.69,Z 332.425,A -85,B 0,C 180,E1 -6527.476,E2 -6527.476} C_VEL
LIN {X 0,Y 488.728,Z 332.421,A -85,B 0,C 180,E1 -6529.678,E2 -6529.678} C_VEL
LIN {X 0,Y 488.679,Z 332.427,A -85,B 0,C 180,E1 -6532.843,E2 -6532.843} C_VEL
LIN {X 0,Y 488.743,Z 332.499,A -85,B 0,C 180,E1 -6534.32,E2 -6534.32} C_VEL
LIN {X 0,Y 489.576,Z 337.373,A -85,B 0,C 180,E1 -6536.368,E2 -6536.368} C_VEL
LIN {X 0,Y 489.732,Z 341.282,A -85,B 0,C 180,E1 -6537.93,E2 -6537.93} C_VEL
LIN {X 0,Y 489.334,Z 349.792,A -85,B 0,C 180,E1 -6541.176,E2 -6541.176} C_VEL
LIN {X 0,Y 488.951,Z 358.701,A -85,B 0,C 180,E1 -6544.457,E2 -6544.457} C_VEL
LIN {X 0,Y 488.734,Z 366.244,A -85,B 0,C 180,E1 -6547.155,E2 -6547.155} C_VEL
LIN {X 0,Y 488.505,Z 375.062,A -85,B 0,C 180,E1 -6550.241,E2 -6550.241} C_VEL
LIN {X 0,Y 488.307,Z 385.196,A -85,B 0,C 180,E1 -6553.702,E2 -6553.702} C_VEL
LIN {X 0,Y 488.126,Z 394.057,A -85,B 0,C 180,E1 -6556.683,E2 -6556.683} C_VEL
LIN {X 0,Y 488.105,Z 399.216,A -85,B 0,C 180,E1 -6558.399,E2 -6558.399} C_VEL
LIN {X 0,Y 489.418,Z 412.012,A -85,B 0,C 180,E1 -6558.823,E2 -6558.823} C_VEL
LIN {X 0,Y 489.374,Z 421.099,A -85,B 0,C 180,E1 -6559.241,E2 -6559.241} C_VEL
LIN {X 0,Y 489.161,Z 429.846,A -85,B 0,C 180,E1 -6559.76,E2 -6559.76} C_VEL
LIN {X 0,Y 488.94,Z 438.203,A -85,B 0,C 180,E1 -6560.382,E2 -6560.382} C_VEL
LIN {X 0,Y 488.669,Z 446.113,A -85,B 0,C 180,E1 -6561.107,E2 -6561.107} C_VEL
LIN {X 0,Y 488.439,Z 453.512,A -85,B 0,C 180,E1 -6561.937,E2 -6561.937} C_VEL
LIN {X 0,Y 488.218,Z 461.023,A -85,B 0,C 180,E1 -6562.973,E2 -6562.973} C_VEL
LIN {X 0,Y 488.123,Z 467.894,A -85,B 0,C 180,E1 -6564.217,E2 -6564.217} C_VEL
LIN {X 0,Y 487.952,Z 473.097,A -85,B 0,C 180,E1 -6565.458,E2 -6565.458} C_VEL
LIN {X 0,Y 487.985,Z 476.923,A -85,B 0,C 180,E1 -6566.699,E2 -6566.699} C_VEL
LIN {X 0,Y 487.935,Z 478.681,A -85,B 0,C 180,E1 -6567.525,E2 -6567.525} C_VEL
LIN {X 0,Y 487.891,Z 479.938,A -85,B 0,C 180,E1 -6568.35,E2 -6568.35} C_VEL
LIN {X 0,Y 487.832,Z 480.717,A -85,B 0,C 180,E1 -6569.176,E2 -6569.176} C_VEL
LIN {X 0,Y 487.82,Z 481.006,A -85,B 0,C 180,E1 -6570.001,E2 -6570.001} C_VEL
LIN {X 0,Y 487.832,Z 480.702,A -85,B 0,C 180,E1 -6570.827,E2 -6570.827} C_VEL
LIN {X 0,Y 487.891,Z 479.91,A -85,B 0,C 180,E1 -6571.652,E2 -6571.652} C_VEL
LIN {X 0,Y 487.936,Z 478.64,A -85,B 0,C 180,E1 -6572.478,E2 -6572.478} C_VEL
LIN {X 0,Y 488.005,Z 475.7,A -85,B 0,C 180,E1 -6573.717,E2 -6573.717} C_VEL
LIN {X 0,Y 487.952,Z 473.018,A -85,B 0,C 180,E1 -6574.545,E2 -6574.545} C_VEL
LIN {X 0,Y 488.124,Z 467.786,A -85,B 0,C 180,E1 -6575.785,E2 -6575.785} C_VEL
LIN {X 0,Y 488.277,Z 460.887,A -85,B 0,C 180,E1 -6577.028,E2 -6577.028} C_VEL
LIN {X 0,Y 488.435,Z 453.355,A -85,B 0,C 180,E1 -6578.066,E2 -6578.066} C_VEL
LIN {X 0,Y 488.671,Z 445.935,A -85,B 0,C 180,E1 -6578.895,E2 -6578.895} C_VEL
LIN {X 0,Y 488.943,Z 437.996,A -85,B 0,C 180,E1 -6579.62,E2 -6579.62} C_VEL
LIN {X 0,Y 489.154,Z 429.614,A -85,B 0,C 180,E1 -6580.243,E2 -6580.243} C_VEL
LIN {X 0,Y 489.455,Z 418.91,A -85,B 0,C 180,E1 -6580.864,E2 -6580.864} C_VEL
LIN {X 0,Y 489.413,Z 411.734,A -85,B 0,C 180,E1 -6581.179,E2 -6581.179} C_VEL
LIN {X 0,Y 488.104,Z 398.835,A -85,B 0,C 180,E1 -6581.63,E2 -6581.63} C_VEL
LIN {X 0,Y 488.256,Z 388.639,A -85,B 0,C 180,E1 -6585.017,E2 -6585.017} C_VEL
LIN {X 0,Y 488.4,Z 378.416,A -85,B 0,C 180,E1 -6588.457,E2 -6588.457} C_VEL
LIN {X 0,Y 488.542,Z 370.773,A -85,B 0,C 180,E1 -6591.079,E2 -6591.079} C_VEL
LIN {X 0,Y 488.727,Z 363.242,A -85,B 0,C 180,E1 -6593.745,E2 -6593.745} C_VEL
LIN {X 0,Y 488.981,Z 355.782,A -85,B 0,C 180,E1 -6596.46,E2 -6596.46} C_VEL
LIN {X 0,Y 489.415,Z 347.177,A -85,B 0,C 180,E1 -6599.698,E2 -6599.698} C_VEL
LIN {X 0,Y 489.733,Z 339.96,A -85,B 0,C 180,E1 -6602.558,E2 -6602.558} C_VEL
LIN {X 0,Y 489.23,Z 335.345,A -85,B 0,C 180,E1 -6604.529,E2 -6604.529} C_VEL
LIN {X 0,Y 488.726,Z 332.423,A -85,B 0,C 180,E1 -6605.874,E2 -6605.874} C_VEL
LIN {X 0,Y 488.706,Z 332.427,A -85,B 0,C 180,E1 -6609.255,E2 -6609.255} C_VEL
LIN {X 0,Y 488.713,Z 332.429,A -85,B 0,C 180,E1 -6611.6,E2 -6611.6} C_VEL
LIN {X 0,Y 488.708,Z 332.426,A -85,B 0,C 180,E1 -6614.803,E2 -6614.803} C_VEL
LIN {X 0,Y 488.698,Z 332.427,A -85,B 0,C 180,E1 -6617.475,E2 -6617.475} C_VEL
LIN {X 0,Y 488.74,Z 332.42,A -85,B 0,C 180,E1 -6619.677,E2 -6619.677} C_VEL
LIN {X 0,Y 488.685,Z 332.426,A -85,B 0,C 180,E1 -6622.841,E2 -6622.841} C_VEL
LIN {X 0,Y 488.73,Z 332.422,A -85,B 0,C 180,E1 -6625.887,E2 -6625.887} C_VEL
LIN {X 0,Y 488.697,Z 332.424,A -85,B 0,C 180,E1 -6628.82,E2 -6628.82} C_VEL
LIN {X 0,Y 488.749,Z 332.42,A -85,B 0,C 180,E1 -6631.671,E2 -6631.671} C_VEL
LIN {X 0,Y 488.747,Z 332.419,A -85,B 0,C 180,E1 -6634.444,E2 -6634.444} C_VEL
LIN {X 0,Y 488.729,Z 332.42,A -85,B 0,C 180,E1 -6637.153,E2 -6637.153} C_VEL
LIN {X 0,Y 488.731,Z 332.421,A -85,B 0,C 180,E1 -6639.81,E2 -6639.81} C_VEL
LIN {X 0,Y 488.72,Z 332.423,A -85,B 0,C 180,E1 -6642.422,E2 -6642.422} C_VEL
LIN {X 0,Y 488.768,Z 332.417,A -85,B 0,C 180,E1 -6644.999,E2 -6644.999} C_VEL
LIN {X 0,Y 488.812,Z 332.412,A -85,B 0,C 180,E1 -6648.387,E2 -6648.387} C_VEL
LIN {X 0,Y 488.791,Z 332.415,A -85,B 0,C 180,E1 -6651.732,E2 -6651.732} C_VEL
LIN {X 0,Y 488.844,Z 332.409,A -85,B 0,C 180,E1 -6654.223,E2 -6654.223} C_VEL
LIN {X 0,Y 488.958,Z 332.394,A -85,B 0,C 180,E1 -6657.528,E2 -6657.528} C_VEL
LIN {X 0,Y 488.94,Z 332.394,A -85,B 0,C 180,E1 -6660.823,E2 -6660.823} C_VEL
LIN {X 0,Y 488.963,Z 332.394,A -85,B 0,C 180,E1 -6662.471,E2 -6662.471} C_VEL
LIN {X 0,Y 488.854,Z 332.406,A -85,B 0,C 180,E1 -6665.775,E2 -6665.775} C_VEL
LIN {X 0,Y 488.788,Z 332.416,A -85,B 0,C 180,E1 -6668.266,E2 -6668.266} C_VEL
LIN {X 0,Y 488.809,Z 332.412,A -85,B 0,C 180,E1 -6671.611,E2 -6671.611} C_VEL
LIN {X 0,Y 488.765,Z 332.418,A -85,B 0,C 180,E1 -6674.999,E2 -6674.999} C_VEL
LIN {X 0,Y 488.661,Z 332.432,A -85,B 0,C 180,E1 -6677.578,E2 -6677.578} C_VEL
LIN {X 0,Y 488.436,Z 332.46,A -85,B 0,C 180,E1 -6679.325,E2 -6679.325} C_VEL
LIN {X 0,Y 488.322,Z 335.689,A -85,B 0,C 180,E1 -6681.973,E2 -6681.973} C_VEL
LIN {X 0,Y 488.278,Z 339.456,A -85,B 0,C 180,E1 -6684.934,E2 -6684.934} C_VEL
LIN {X 0,Y 488.176,Z 343.886,A -85,B 0,C 180,E1 -6688.363,E2 -6688.363} C_VEL
LIN {X 0,Y 488.072,Z 347.644,A -85,B 0,C 180,E1 -6691.222,E2 -6691.222} C_VEL
LIN {X 0,Y 488.025,Z 351.552,A -85,B 0,C 180,E1 -6694.167,E2 -6694.167} C_VEL
LIN {X 0,Y 487.942,Z 355.665,A -85,B 0,C 180,E1 -6697.223,E2 -6697.223} C_VEL
LIN {X 0,Y 487.965,Z 357.435,A -85,B 0,C 180,E1 -6698.513,E2 -6698.513} C_VEL
LIN {X 0,Y 489.687,Z 367.705,A -85,B 0,C 180,E1 -6698.909,E2 -6698.909} C_VEL
LIN {X 0,Y 489.59,Z 376.94,A -85,B 0,C 180,E1 -6699.347,E2 -6699.347} C_VEL
LIN {X 0,Y 489.385,Z 385.271,A -85,B 0,C 180,E1 -6699.854,E2 -6699.854} C_VEL
LIN {X 0,Y 489.127,Z 393.399,A -85,B 0,C 180,E1 -6700.47,E2 -6700.47} C_VEL
LIN {X 0,Y 488.933,Z 400.537,A -85,B 0,C 180,E1 -6701.132,E2 -6701.132} C_VEL
LIN {X 0,Y 488.707,Z 407.498,A -85,B 0,C 180,E1 -6701.911,E2 -6701.911} C_VEL
LIN {X 0,Y 488.507,Z 414.017,A -85,B 0,C 180,E1 -6702.8,E2 -6702.8} C_VEL
LIN {X 0,Y 488.263,Z 420.924,A -85,B 0,C 180,E1 -6703.97,E2 -6703.97} C_VEL
LIN {X 0,Y 488.127,Z 426.072,A -85,B 0,C 180,E1 -6705.129,E2 -6705.129} C_VEL
LIN {X 0,Y 488.016,Z 429.888,A -85,B 0,C 180,E1 -6706.269,E2 -6706.269} C_VEL
LIN {X 0,Y 487.939,Z 432.583,A -85,B 0,C 180,E1 -6707.392,E2 -6707.392} C_VEL
LIN {X 0,Y 487.885,Z 434.292,A -85,B 0,C 180,E1 -6708.507,E2 -6708.507} C_VEL
LIN {X 0,Y 487.846,Z 435.14,A -85,B 0,C 180,E1 -6709.774,E2 -6709.774} C_VEL
LIN {X 0,Y 487.82,Z 434.824,A -85,B 0,C 180,E1 -6711.073,E2 -6711.073} C_VEL
LIN {X 0,Y 487.861,Z 433.125,A -85,B 0,C 180,E1 -6712.4,E2 -6712.4} C_VEL
LIN {X 0,Y 487.983,Z 431.284,A -85,B 0,C 180,E1 -6713.295,E2 -6713.295} C_VEL
LIN {X 0,Y 488.04,Z 428.326,A -85,B 0,C 180,E1 -6714.322,E2 -6714.322} C_VEL
LIN {X 0,Y 488.151,Z 423.723,A -85,B 0,C 180,E1 -6715.498,E2 -6715.498} C_VEL
LIN {X 0,Y 488.329,Z 418.221,A -85,B 0,C 180,E1 -6716.586,E2 -6716.586} C_VEL
LIN {X 0,Y 488.477,Z 413.719,A -85,B 0,C 180,E1 -6717.316,E2 -6717.316} C_VEL
LIN {X 0,Y 487.924,Z 410.146,A -85,B 0,C 180,E1 -6717.849,E2 -6717.849} C_VEL
LIN {X 0,Y 485.289,Z 403.793,A -85,B 0,C 180,E1 -6718.686,E2 -6718.686} C_VEL
LIN {X 0,Y 482.672,Z 396.758,A -85,B 0,C 180,E1 -6719.465,E2 -6719.465} C_VEL
LIN {X 0,Y 482.154,Z 391.97,A -85,B 0,C 180,E1 -6719.892,E2 -6719.892} C_VEL
LIN {X 0,Y 482.443,Z 381.695,A -85,B 0,C 180,E1 -6720.635,E2 -6720.635} C_VEL
LIN {X 0,Y 482.734,Z 371.273,A -85,B 0,C 180,E1 -6721.186,E2 -6721.186} C_VEL
LIN {X 0,Y 482.404,Z 365.619,A -85,B 0,C 180,E1 -6721.442,E2 -6721.442} C_VEL
LIN {X 0,Y 480.89,Z 357.363,A -85,B 0,C 180,E1 -6721.76,E2 -6721.76} C_VEL
LIN {X 0,Y 480.944,Z 353.003,A -85,B 0,C 180,E1 -6724.955,E2 -6724.955} C_VEL
LIN {X 0,Y 480.94,Z 349.345,A -85,B 0,C 180,E1 -6727.669,E2 -6727.669} C_VEL
LIN {X 0,Y 481.003,Z 345.754,A -85,B 0,C 180,E1 -6730.362,E2 -6730.362} C_VEL
LIN {X 0,Y 481.065,Z 342.262,A -85,B 0,C 180,E1 -6733.01,E2 -6733.01} C_VEL
LIN {X 0,Y 481.117,Z 338.857,A -85,B 0,C 180,E1 -6735.62,E2 -6735.62} C_VEL
LIN {X 0,Y 481.308,Z 334.39,A -85,B 0,C 180,E1 -6739.056,E2 -6739.056} C_VEL
LIN {X 0,Y 481.283,Z 333.35,A -85,B 0,C 180,E1 -6739.907,E2 -6739.907} C_VEL
LIN {X 0,Y 481.751,Z 333.289,A -85,B 0,C 180,E1 -6742.742,E2 -6742.742} C_VEL
LIN {X 0,Y 481.772,Z 333.286,A -85,B 0,C 180,E1 -6744.978,E2 -6744.978} C_VEL
LIN {X 0,Y 481.918,Z 333.27,A -85,B 0,C 180,E1 -6747.491,E2 -6747.491} C_VEL
LIN {X 0,Y 481.929,Z 333.268,A -85,B 0,C 180,E1 -6749.999,E2 -6749.999} C_VEL
LIN {X 0,Y 481.919,Z 333.268,A -85,B 0,C 180,E1 -6752.506,E2 -6752.506} C_VEL
LIN {X 0,Y 481.818,Z 333.283,A -85,B 0,C 180,E1 -6755.859,E2 -6755.859} C_VEL
LIN {X 0,Y 481.752,Z 333.289,A -85,B 0,C 180,E1 -6758.387,E2 -6758.387} C_VEL
LIN {X 0,Y 481.783,Z 333.288,A -85,B 0,C 180,E1 -6761.783,E2 -6761.783} C_VEL
LIN {X 0,Y 481.729,Z 333.292,A -85,B 0,C 180,E1 -6765.223,E2 -6765.223} C_VEL
LIN {X 0,Y 481.699,Z 333.295,A -85,B 0,C 180,E1 -6768.721,E2 -6768.721} C_VEL
LIN {X 0,Y 481.634,Z 333.306,A -85,B 0,C 180,E1 -6771.394,E2 -6771.394} C_VEL
LIN {X 0,Y 481.663,Z 333.3,A -85,B 0,C 180,E1 -6774.112,E2 -6774.112} C_VEL
LIN {X 0,Y 481.738,Z 333.291,A -85,B 0,C 180,E1 -6777.14,E2 -6777.14} C_VEL
LIN {X 0,Y 481.674,Z 333.301,A -85,B 0,C 180,E1 -6779.74,E2 -6779.74} C_VEL
LIN {X 0,Y 481.659,Z 333.302,A -85,B 0,C 180,E1 -6782.674,E2 -6782.674} C_VEL
LIN {X 0,Y 481.629,Z 333.306,A -85,B 0,C 180,E1 -6785.708,E2 -6785.708} C_VEL
LIN {X 0,Y 481.705,Z 333.297,A -85,B 0,C 180,E1 -6789.354,E2 -6789.354} C_VEL
LIN {X 0,Y 481.66,Z 333.301,A -85,B 0,C 180,E1 -6792.157,E2 -6792.157} C_VEL
LIN {X 0,Y 481.645,Z 333.303,A -85,B 0,C 180,E1 -6794.457,E2 -6794.457} C_VEL
LIN {X 0,Y 481.674,Z 333.301,A -85,B 0,C 180,E1 -6796.846,E2 -6796.846} C_VEL
LIN {X 0,Y 481.677,Z 333.297,A -85,B 0,C 180,E1 -6800.061,E2 -6800.061} C_VEL
LIN {X 0,Y 481.617,Z 333.306,A -85,B 0,C 180,E1 -6803.254,E2 -6803.254} C_VEL
LIN {X 0,Y 481.694,Z 333.297,A -85,B 0,C 180,E1 -6806.33,E2 -6806.33} C_VEL
LIN {X 0,Y 481.644,Z 333.302,A -85,B 0,C 180,E1 -6809.416,E2 -6809.416} C_VEL
LIN {X 0,Y 481.687,Z 333.298,A -85,B 0,C 180,E1 -6812.169,E2 -6812.169} C_VEL
LIN {X 0,Y 481.708,Z 333.297,A -85,B 0,C 180,E1 -6814.971,E2 -6814.971} C_VEL
LIN {X 0,Y 481.647,Z 333.303,A -85,B 0,C 180,E1 -6817.706,E2 -6817.706} C_VEL
LIN {X 0,Y 481.695,Z 333.298,A -85,B 0,C 180,E1 -6820.394,E2 -6820.394} C_VEL
LIN {X 0,Y 481.679,Z 333.298,A -85,B 0,C 180,E1 -6823.035,E2 -6823.035} C_VEL
LIN {X 0,Y 481.677,Z 333.298,A -85,B 0,C 180,E1 -6825.639,E2 -6825.639} C_VEL
LIN {X 0,Y 481.782,Z 333.287,A -85,B 0,C 180,E1 -6828.217,E2 -6828.217} C_VEL
LIN {X 0,Y 481.751,Z 333.289,A -85,B 0,C 180,E1 -6831.612,E2 -6831.612} C_VEL
LIN {X 0,Y 481.806,Z 333.283,A -85,B 0,C 180,E1 -6834.14,E2 -6834.14} C_VEL
LIN {X 0,Y 481.919,Z 333.269,A -85,B 0,C 180,E1 -6837.493,E2 -6837.493} C_VEL
LIN {X 0,Y 481.916,Z 333.269,A -85,B 0,C 180,E1 -6840.836,E2 -6840.836} C_VEL
LIN {X 0,Y 481.919,Z 333.268,A -85,B 0,C 180,E1 -6842.508,E2 -6842.508} C_VEL
LIN {X 0,Y 481.806,Z 333.284,A -85,B 0,C 180,E1 -6845.861,E2 -6845.861} C_VEL
LIN {X 0,Y 481.753,Z 333.288,A -85,B 0,C 180,E1 -6848.389,E2 -6848.389} C_VEL
LIN {X 0,Y 481.785,Z 333.287,A -85,B 0,C 180,E1 -6851.785,E2 -6851.785} C_VEL
LIN {X 0,Y 481.733,Z 333.293,A -85,B 0,C 180,E1 -6855.225,E2 -6855.225} C_VEL
LIN {X 0,Y 481.703,Z 333.295,A -85,B 0,C 180,E1 -6858.723,E2 -6858.723} C_VEL
LIN {X 0,Y 481.638,Z 333.306,A -85,B 0,C 180,E1 -6861.396,E2 -6861.396} C_VEL
LIN {X 0,Y 481.669,Z 333.298,A -85,B 0,C 180,E1 -6864.114,E2 -6864.114} C_VEL
LIN {X 0,Y 481.744,Z 333.291,A -85,B 0,C 180,E1 -6867.142,E2 -6867.142} C_VEL
LIN {X 0,Y 481.68,Z 333.3,A -85,B 0,C 180,E1 -6869.742,E2 -6869.742} C_VEL
LIN {X 0,Y 481.665,Z 333.301,A -85,B 0,C 180,E1 -6872.675,E2 -6872.675} C_VEL
LIN {X 0,Y 481.636,Z 333.305,A -85,B 0,C 180,E1 -6875.71,E2 -6875.71} C_VEL
LIN {X 0,Y 481.664,Z 333.301,A -85,B 0,C 180,E1 -6878.86,E2 -6878.86} C_VEL
LIN {X 0,Y 481.656,Z 333.302,A -85,B 0,C 180,E1 -6881.915,E2 -6881.915} C_VEL
LIN {X 0,Y 481.654,Z 333.303,A -85,B 0,C 180,E1 -6884.458,E2 -6884.458} C_VEL
LIN {X 0,Y 481.649,Z 333.302,A -85,B 0,C 180,E1 -6887.841,E2 -6887.841} C_VEL
LIN {X 0,Y 481.676,Z 333.3,A -85,B 0,C 180,E1 -6890.652,E2 -6890.652} C_VEL
LIN {X 0,Y 481.711,Z 333.47,A -85,B 0,C 180,E1 -6894.17,E2 -6894.17} C_VEL
LIN {X 0,Y 482.61,Z 338.712,A -85,B 0,C 180,E1 -6896.403,E2 -6896.403} C_VEL
LIN {X 0,Y 482.748,Z 341.672,A -85,B 0,C 180,E1 -6897.606,E2 -6897.606} C_VEL
LIN {X 0,Y 482.33,Z 350.278,A -85,B 0,C 180,E1 -6900.958,E2 -6900.958} C_VEL
LIN {X 0,Y 481.983,Z 358.527,A -85,B 0,C 180,E1 -6904.061,E2 -6904.061} C_VEL
LIN {X 0,Y 481.71,Z 366.041,A -85,B 0,C 180,E1 -6906.803,E2 -6906.803} C_VEL
LIN {X 0,Y 481.418,Z 376.107,A -85,B 0,C 180,E1 -6910.382,E2 -6910.382} C_VEL
LIN {X 0,Y 481.236,Z 386.204,A -85,B 0,C 180,E1 -6913.892,E2 -6913.892} C_VEL
LIN {X 0,Y 481.032,Z 395.046,A -85,B 0,C 180,E1 -6916.913,E2 -6916.913} C_VEL
LIN {X 0,Y 481.015,Z 398.904,A -85,B 0,C 180,E1 -6918.216,E2 -6918.216} C_VEL
LIN {X 0,Y 482.392,Z 412.129,A -85,B 0,C 180,E1 -6918.68,E2 -6918.68} C_VEL
LIN {X 0,Y 482.379,Z 420.737,A -85,B 0,C 180,E1 -6919.083,E2 -6919.083} C_VEL
LIN {X 0,Y 482.174,Z 429.491,A -85,B 0,C 180,E1 -6919.61,E2 -6919.61} C_VEL
LIN {X 0,Y 481.905,Z 437.852,A -85,B 0,C 180,E1 -6920.24,E2 -6920.24} C_VEL
LIN {X 0,Y 481.618,Z 445.766,A -85,B 0,C 180,E1 -6920.976,E2 -6920.976} C_VEL
LIN {X 0,Y 481.395,Z 453.17,A -85,B 0,C 180,E1 -6921.818,E2 -6921.818} C_VEL
LIN {X 0,Y 481.157,Z 460.684,A -85,B 0,C 180,E1 -6922.869,E2 -6922.869} C_VEL
LIN {X 0,Y 481.025,Z 467.559,A -85,B 0,C 180,E1 -6924.131,E2 -6924.131} C_VEL
LIN {X 0,Y 480.87,Z 472.764,A -85,B 0,C 180,E1 -6925.391,E2 -6925.391} C_VEL
LIN {X 0,Y 480.914,Z 476.592,A -85,B 0,C 180,E1 -6926.65,E2 -6926.65} C_VEL
LIN {X 0,Y 480.848,Z 478.349,A -85,B 0,C 180,E1 -6927.488,E2 -6927.488} C_VEL
LIN {X 0,Y 480.822,Z 479.608,A -85,B 0,C 180,E1 -6928.326,E2 -6928.326} C_VEL
LIN {X 0,Y 480.758,Z 480.386,A -85,B 0,C 180,E1 -6929.163,E2 -6929.163} C_VEL
LIN {X 0,Y 480.744,Z 480.674,A -85,B 0,C 180,E1 -6930.001,E2 -6930.001} C_VEL
LIN {X 0,Y 480.758,Z 480.368,A -85,B 0,C 180,E1 -6930.839,E2 -6930.839} C_VEL
LIN {X 0,Y 480.823,Z 479.575,A -85,B 0,C 180,E1 -6931.676,E2 -6931.676} C_VEL
LIN {X 0,Y 480.849,Z 478.301,A -85,B 0,C 180,E1 -6932.514,E2 -6932.514} C_VEL
LIN {X 0,Y 480.925,Z 475.359,A -85,B 0,C 180,E1 -6933.772,E2 -6933.772} C_VEL
LIN {X 0,Y 480.87,Z 472.674,A -85,B 0,C 180,E1 -6934.612,E2 -6934.612} C_VEL
LIN {X 0,Y 481.026,Z 467.438,A -85,B 0,C 180,E1 -6935.871,E2 -6935.871} C_VEL
LIN {X 0,Y 481.208,Z 460.535,A -85,B 0,C 180,E1 -6937.132,E2 -6937.132} C_VEL
LIN {X 0,Y 481.383,Z 453,A -85,B 0,C 180,E1 -6938.185,E2 -6938.185} C_VEL
LIN {X 0,Y 481.619,Z 445.577,A -85,B 0,C 180,E1 -6939.026,E2 -6939.026} C_VEL
LIN {X 0,Y 481.888,Z 437.636,A -85,B 0,C 180,E1 -6939.762,E2 -6939.762} C_VEL
LIN {X 0,Y 482.211,Z 427.75,A -85,B 0,C 180,E1 -6940.498,E2 -6940.498} C_VEL
LIN {X 0,Y 482.544,Z 416.478,A -85,B 0,C 180,E1 -6941.116,E2 -6941.116} C_VEL
LIN {X 0,Y 481.931,Z 407.901,A -85,B 0,C 180,E1 -6941.482,E2 -6941.482} C_VEL
LIN {X 0,Y 481.017,Z 398.55,A -85,B 0,C 180,E1 -6941.785,E2 -6941.785} C_VEL
LIN {X 0,Y 481.173,Z 388.325,A -85,B 0,C 180,E1 -6945.244,E2 -6945.244} C_VEL
LIN {X 0,Y 481.36,Z 378.157,A -85,B 0,C 180,E1 -6948.737,E2 -6948.737} C_VEL
LIN {X 0,Y 481.546,Z 369.296,A -85,B 0,C 180,E1 -6951.85,E2 -6951.85} C_VEL
LIN {X 0,Y 481.848,Z 360.546,A -85,B 0,C 180,E1 -6955.024,E2 -6955.024} C_VEL
LIN {X 0,Y 482.159,Z 351.95,A -85,B 0,C 180,E1 -6958.277,E2 -6958.277} C_VEL
LIN {X 0,Y 482.517,Z 345.63,A -85,B 0,C 180,E1 -6960.756,E2 -6960.756} C_VEL
LIN {X 0,Y 482.762,Z 339.905,A -85,B 0,C 180,E1 -6963.089,E2 -6963.089} C_VEL
LIN {X 0,Y 481.692,Z 333.505,A -85,B 0,C 180,E1 -6965.964,E2 -6965.964} C_VEL
LIN {X 0,Y 481.686,Z 333.303,A -85,B 0,C 180,E1 -6969.349,E2 -6969.349} C_VEL
LIN {X 0,Y 481.654,Z 333.306,A -85,B 0,C 180,E1 -6972.161,E2 -6972.161} C_VEL
LIN {X 0,Y 481.661,Z 333.304,A -85,B 0,C 180,E1 -6975.542,E2 -6975.542} C_VEL
LIN {X 0,Y 481.663,Z 333.303,A -85,B 0,C 180,E1 -6978.958,E2 -6978.958} C_VEL
LIN {X 0,Y 481.66,Z 333.302,A -85,B 0,C 180,E1 -6981.993,E2 -6981.993} C_VEL
LIN {X 0,Y 481.691,Z 333.297,A -85,B 0,C 180,E1 -6985.318,E2 -6985.318} C_VEL
LIN {X 0,Y 481.651,Z 333.304,A -85,B 0,C 180,E1 -6988.311,E2 -6988.311} C_VEL
LIN {X 0,Y 481.704,Z 333.295,A -85,B 0,C 180,E1 -6991.218,E2 -6991.218} C_VEL
LIN {X 0,Y 481.704,Z 333.298,A -85,B 0,C 180,E1 -6994.042,E2 -6994.042} C_VEL
LIN {X 0,Y 481.681,Z 333.299,A -85,B 0,C 180,E1 -6996.812,E2 -6996.812} C_VEL
LIN {X 0,Y 481.702,Z 333.296,A -85,B 0,C 180,E1 -6999.502,E2 -6999.502} C_VEL
LIN {X 0,Y 481.698,Z 333.297,A -85,B 0,C 180,E1 -7002.157,E2 -7002.157} C_VEL
LIN {X 0,Y 481.749,Z 333.292,A -85,B 0,C 180,E1 -7004.775,E2 -7004.775} C_VEL
LIN {X 0,Y 481.757,Z 333.291,A -85,B 0,C 180,E1 -7008.215,E2 -7008.215} C_VEL
LIN {X 0,Y 481.745,Z 333.292,A -85,B 0,C 180,E1 -7011.611,E2 -7011.611} C_VEL
LIN {X 0,Y 481.803,Z 333.285,A -85,B 0,C 180,E1 -7014.139,E2 -7014.139} C_VEL
LIN {X 0,Y 481.925,Z 333.269,A -85,B 0,C 180,E1 -7017.492,E2 -7017.492} C_VEL
LIN {X 0,Y 481.892,Z 333.272,A -85,B 0,C 180,E1 -7020.835,E2 -7020.835} C_VEL
LIN {X 0,Y 481.93,Z 333.269,A -85,B 0,C 180,E1 -7022.507,E2 -7022.507} C_VEL
LIN {X 0,Y 481.815,Z 333.283,A -85,B 0,C 180,E1 -7025.86,E2 -7025.86} C_VEL
LIN {X 0,Y 481.743,Z 333.293,A -85,B 0,C 180,E1 -7028.388,E2 -7028.388} C_VEL
LIN {X 0,Y 481.755,Z 333.292,A -85,B 0,C 180,E1 -7031.784,E2 -7031.784} C_VEL
LIN {X 0,Y 481.746,Z 333.294,A -85,B 0,C 180,E1 -7035.223,E2 -7035.223} C_VEL
LIN {X 0,Y 481.609,Z 333.311,A -85,B 0,C 180,E1 -7037.844,E2 -7037.844} C_VEL
LIN {X 0,Y 481.363,Z 333.525,A -85,B 0,C 180,E1 -7039.62,E2 -7039.62} C_VEL
LIN {X 0,Y 481.268,Z 337.856,A -85,B 0,C 180,E1 -7043.073,E2 -7043.073} C_VEL
LIN {X 0,Y 481.139,Z 341.524,A -85,B 0,C 180,E1 -7045.988,E2 -7045.988} C_VEL
LIN {X 0,Y 481.096,Z 345.196,A -85,B 0,C 180,E1 -7048.82,E2 -7048.82} C_VEL
LIN {X 0,Y 480.996,Z 349.417,A -85,B 0,C 180,E1 -7052.063,E2 -7052.063} C_VEL
LIN {X 0,Y 480.912,Z 353.38,A -85,B 0,C 180,E1 -7055.076,E2 -7055.076} C_VEL
LIN {X 0,Y 480.862,Z 357.713,A -85,B 0,C 180,E1 -7058.316,E2 -7058.316} C_VEL
LIN {X 0,Y 482.711,Z 368.34,A -85,B 0,C 180,E1 -7058.758,E2 -7058.758} C_VEL
LIN {X 0,Y 482.625,Z 377.702,A -85,B 0,C 180,E1 -7059.215,E2 -7059.215} C_VEL
LIN {X 0,Y 482.418,Z 386.252,A -85,B 0,C 180,E1 -7059.751,E2 -7059.751} C_VEL
LIN {X 0,Y 482.151,Z 393.396,A -85,B 0,C 180,E1 -7060.301,E2 -7060.301} C_VEL
LIN {X 0,Y 481.94,Z 400.961,A -85,B 0,C 180,E1 -7061.011,E2 -7061.011} C_VEL
LIN {X 0,Y 481.707,Z 407.498,A -85,B 0,C 180,E1 -7061.75,E2 -7061.75} C_VEL
LIN {X 0,Y 481.485,Z 414.016,A -85,B 0,C 180,E1 -7062.643,E2 -7062.643} C_VEL
LIN {X 0,Y 481.271,Z 419.592,A -85,B 0,C 180,E1 -7063.575,E2 -7063.575} C_VEL
LIN {X 0,Y 481.115,Z 425.248,A -85,B 0,C 180,E1 -7064.756,E2 -7064.756} C_VEL
LIN {X 0,Y 480.996,Z 428.785,A -85,B 0,C 180,E1 -7065.72,E2 -7065.72} C_VEL
LIN {X 0,Y 480.899,Z 432.136,A -85,B 0,C 180,E1 -7066.944,E2 -7066.944} C_VEL
LIN {X 0,Y 480.798,Z 434.305,A -85,B 0,C 180,E1 -7068.199,E2 -7068.199} C_VEL
LIN {X 0,Y 480.796,Z 435.06,A -85,B 0,C 180,E1 -7068.868,E2 -7068.868} C_VEL
LIN {X 0,Y 480.743,Z 435.542,A -85,B 0,C 180,E1 -7069.965,E2 -7069.965} C_VEL
LIN {X 0,Y 480.752,Z 435.177,A -85,B 0,C 180,E1 -7071.052,E2 -7071.052} C_VEL
LIN {X 0,Y 480.784,Z 433.994,A -85,B 0,C 180,E1 -7072.124,E2 -7072.124} C_VEL
LIN {X 0,Y 480.903,Z 431.206,A -85,B 0,C 180,E1 -7073.49,E2 -7073.49} C_VEL
LIN {X 0,Y 480.987,Z 427.872,A -85,B 0,C 180,E1 -7074.599,E2 -7074.599} C_VEL
LIN {X 0,Y 481.098,Z 424.289,A -85,B 0,C 180,E1 -7075.522,E2 -7075.522} C_VEL
LIN {X 0,Y 481.28,Z 419.054,A -85,B 0,C 180,E1 -7076.588,E2 -7076.588} C_VEL
LIN {X 0,Y 481.447,Z 413.817,A -85,B 0,C 180,E1 -7077.454,E2 -7077.454} C_VEL
LIN {X 0,Y 481.722,Z 406.505,A -85,B 0,C 180,E1 -7078.439,E2 -7078.439} C_VEL
LIN {X 0,Y 481.986,Z 397.353,A -85,B 0,C 180,E1 -7079.427,E2 -7079.427} C_VEL
LIN {X 0,Y 482.154,Z 391.97,A -85,B 0,C 180,E1 -7079.892,E2 -7079.892} C_VEL
LIN {X 0,Y 481.768,Z 387.126,A -85,B 0,C 180,E1 -7080.294,E2 -7080.294} C_VEL
LIN {X 0,Y 479.515,Z 378.932,A -85,B 0,C 180,E1 -7080.899,E2 -7080.899} C_VEL
LIN {X 0,Y 476.044,Z 368.589,A -85,B 0,C 180,E1 -7081.493,E2 -7081.493} C_VEL
LIN {X 0,Y 475.126,Z 364.933,A -85,B 0,C 180,E1 -7081.651,E2 -7081.651} C_VEL
LIN {X 0,Y 473.826,Z 357.661,A -85,B 0,C 180,E1 -7081.934,E2 -7081.934} C_VEL
LIN {X 0,Y 473.865,Z 353.813,A -85,B 0,C 180,E1 -7084.78,E2 -7084.78} C_VEL
LIN {X 0,Y 473.871,Z 350.41,A -85,B 0,C 180,E1 -7087.318,E2 -7087.318} C_VEL
LIN {X 0,Y 473.916,Z 346.793,A -85,B 0,C 180,E1 -7090.056,E2 -7090.056} C_VEL
LIN {X 0,Y 473.982,Z 343.249,A -85,B 0,C 180,E1 -7092.748,E2 -7092.748} C_VEL
LIN {X 0,Y 474.045,Z 339.824,A -85,B 0,C 180,E1 -7095.401,E2 -7095.401} C_VEL
LIN {X 0,Y 474.252,Z 335.332,A -85,B 0,C 180,E1 -7098.892,E2 -7098.892} C_VEL
LIN {X 0,Y 474.216,Z 334.25,A -85,B 0,C 180,E1 -7099.755,E2 -7099.755} C_VEL
LIN {X 0,Y 474.716,Z 334.166,A -85,B 0,C 180,E1 -7102.695,E2 -7102.695} C_VEL
LIN {X 0,Y 474.742,Z 334.162,A -85,B 0,C 180,E1 -7104.903,E2 -7104.903} C_VEL
LIN {X 0,Y 474.884,Z 334.146,A -85,B 0,C 180,E1 -7107.454,E2 -7107.454} C_VEL
LIN {X 0,Y 474.9,Z 334.144,A -85,B 0,C 180,E1 -7109.999,E2 -7109.999} C_VEL
LIN {X 0,Y 474.885,Z 334.145,A -85,B 0,C 180,E1 -7112.544,E2 -7112.544} C_VEL
LIN {X 0,Y 474.779,Z 334.159,A -85,B 0,C 180,E1 -7115.946,E2 -7115.946} C_VEL
LIN {X 0,Y 474.718,Z 334.165,A -85,B 0,C 180,E1 -7118.513,E2 -7118.513} C_VEL
LIN {X 0,Y 474.727,Z 334.166,A -85,B 0,C 180,E1 -7121.961,E2 -7121.961} C_VEL
LIN {X 0,Y 474.667,Z 334.173,A -85,B 0,C 180,E1 -7125.767,E2 -7125.767} C_VEL
LIN {X 0,Y 474.652,Z 334.174,A -85,B 0,C 180,E1 -7129.009,E2 -7129.009} C_VEL
LIN {X 0,Y 474.577,Z 334.184,A -85,B 0,C 180,E1 -7131.728,E2 -7131.728} C_VEL
LIN {X 0,Y 474.645,Z 334.173,A -85,B 0,C 180,E1 -7134.492,E2 -7134.492} C_VEL
LIN {X 0,Y 474.685,Z 334.171,A -85,B 0,C 180,E1 -7137.338,E2 -7137.338} C_VEL
LIN {X 0,Y 474.595,Z 334.18,A -85,B 0,C 180,E1 -7140.811,E2 -7140.811} C_VEL
LIN {X 0,Y 474.623,Z 334.176,A -85,B 0,C 180,E1 -7143.984,E2 -7143.984} C_VEL
LIN {X 0,Y 474.563,Z 334.185,A -85,B 0,C 180,E1 -7146.9,E2 -7146.9} C_VEL
LIN {X 0,Y 474.64,Z 334.176,A -85,B 0,C 180,E1 -7149.651,E2 -7149.651} C_VEL
LIN {X 0,Y 474.637,Z 334.176,A -85,B 0,C 180,E1 -7152.93,E2 -7152.93} C_VEL
LIN {X 0,Y 474.603,Z 334.18,A -85,B 0,C 180,E1 -7155.896,E2 -7155.896} C_VEL
LIN {X 0,Y 474.63,Z 334.178,A -85,B 0,C 180,E1 -7159.038,E2 -7159.038} C_VEL
LIN {X 0,Y 474.606,Z 334.18,A -85,B 0,C 180,E1 -7161.702,E2 -7161.702} C_VEL
LIN {X 0,Y 474.616,Z 334.179,A -85,B 0,C 180,E1 -7164.726,E2 -7164.726} C_VEL
LIN {X 0,Y 474.623,Z 334.177,A -85,B 0,C 180,E1 -7167.788,E2 -7167.788} C_VEL
LIN {X 0,Y 474.618,Z 334.179,A -85,B 0,C 180,E1 -7170.883,E2 -7170.883} C_VEL
LIN {X 0,Y 474.647,Z 334.174,A -85,B 0,C 180,E1 -7173.629,E2 -7173.629} C_VEL
LIN {X 0,Y 474.623,Z 334.179,A -85,B 0,C 180,E1 -7176.641,E2 -7176.641} C_VEL
LIN {X 0,Y 474.662,Z 334.171,A -85,B 0,C 180,E1 -7179.186,E2 -7179.186} C_VEL
LIN {X 0,Y 474.644,Z 334.175,A -85,B 0,C 180,E1 -7181.885,E2 -7181.885} C_VEL
LIN {X 0,Y 474.686,Z 334.171,A -85,B 0,C 180,E1 -7184.545,E2 -7184.545} C_VEL
LIN {X 0,Y 474.726,Z 334.165,A -85,B 0,C 180,E1 -7188.039,E2 -7188.039} C_VEL
LIN {X 0,Y 474.717,Z 334.165,A -85,B 0,C 180,E1 -7191.487,E2 -7191.487} C_VEL
LIN {X 0,Y 474.768,Z 334.16,A -85,B 0,C 180,E1 -7194.053,E2 -7194.053} C_VEL
LIN {X 0,Y 474.885,Z 334.145,A -85,B 0,C 180,E1 -7197.456,E2 -7197.456} C_VEL
LIN {X 0,Y 474.867,Z 334.147,A -85,B 0,C 180,E1 -7200.849,E2 -7200.849} C_VEL
LIN {X 0,Y 474.886,Z 334.144,A -85,B 0,C 180,E1 -7202.545,E2 -7202.545} C_VEL
LIN {X 0,Y 474.768,Z 334.16,A -85,B 0,C 180,E1 -7205.948,E2 -7205.948} C_VEL
LIN {X 0,Y 474.718,Z 334.164,A -85,B 0,C 180,E1 -7208.514,E2 -7208.514} C_VEL
LIN {X 0,Y 474.729,Z 334.165,A -85,B 0,C 180,E1 -7211.962,E2 -7211.962} C_VEL
LIN {X 0,Y 474.671,Z 334.172,A -85,B 0,C 180,E1 -7215.769,E2 -7215.769} C_VEL
LIN {X 0,Y 474.655,Z 334.175,A -85,B 0,C 180,E1 -7219.011,E2 -7219.011} C_VEL
LIN {X 0,Y 474.581,Z 334.183,A -85,B 0,C 180,E1 -7221.73,E2 -7221.73} C_VEL
LIN {X 0,Y 474.651,Z 334.172,A -85,B 0,C 180,E1 -7224.494,E2 -7224.494} C_VEL
LIN {X 0,Y 474.691,Z 334.172,A -85,B 0,C 180,E1 -7227.34,E2 -7227.34} C_VEL
LIN {X 0,Y 474.601,Z 334.18,A -85,B 0,C 180,E1 -7230.812,E2 -7230.812} C_VEL
LIN {X 0,Y 474.631,Z 334.175,A -85,B 0,C 180,E1 -7233.985,E2 -7233.985} C_VEL
LIN {X 0,Y 474.568,Z 334.185,A -85,B 0,C 180,E1 -7236.901,E2 -7236.901} C_VEL
LIN {X 0,Y 474.621,Z 334.178,A -85,B 0,C 180,E1 -7239.649,E2 -7239.649} C_VEL
LIN {X 0,Y 474.629,Z 334.178,A -85,B 0,C 180,E1 -7242.933,E2 -7242.933} C_VEL
LIN {X 0,Y 474.609,Z 334.179,A -85,B 0,C 180,E1 -7245.897,E2 -7245.897} C_VEL
LIN {X 0,Y 474.627,Z 334.179,A -85,B 0,C 180,E1 -7249.041,E2 -7249.041} C_VEL
LIN {X 0,Y 474.606,Z 334.18,A -85,B 0,C 180,E1 -7251.705,E2 -7251.705} C_VEL
LIN {X 0,Y 474.663,Z 334.3,A -85,B 0,C 180,E1 -7253.957,E2 -7253.957} C_VEL
LIN {X 0,Y 475.611,Z 339.854,A -85,B 0,C 180,E1 -7256.37,E2 -7256.37} C_VEL
LIN {X 0,Y 475.718,Z 343.501,A -85,B 0,C 180,E1 -7257.872,E2 -7257.872} C_VEL
LIN {X 0,Y 475.256,Z 352.145,A -85,B 0,C 180,E1 -7261.277,E2 -7261.277} C_VEL
LIN {X 0,Y 474.852,Z 360.72,A -85,B 0,C 180,E1 -7264.532,E2 -7264.532} C_VEL
LIN {X 0,Y 474.584,Z 368.343,A -85,B 0,C 180,E1 -7267.356,E2 -7267.356} C_VEL
LIN {X 0,Y 474.326,Z 377.133,A -85,B 0,C 180,E1 -7270.527,E2 -7270.527} C_VEL
LIN {X 0,Y 474.152,Z 385.938,A -85,B 0,C 180,E1 -7273.644,E2 -7273.644} C_VEL
LIN {X 0,Y 473.964,Z 394.754,A -85,B 0,C 180,E1 -7276.714,E2 -7276.714} C_VEL
LIN {X 0,Y 473.929,Z 398.623,A -85,B 0,C 180,E1 -7278.05,E2 -7278.05} C_VEL
LIN {X 0,Y 475.184,Z 411.117,A -85,B 0,C 180,E1 -7278.478,E2 -7278.478} C_VEL
LIN {X 0,Y 475.525,Z 416.992,A -85,B 0,C 180,E1 -7278.749,E2 -7278.749} C_VEL
LIN {X 0,Y 475.269,Z 427.63,A -85,B 0,C 180,E1 -7279.349,E2 -7279.349} C_VEL
LIN {X 0,Y 474.858,Z 437.493,A -85,B 0,C 180,E1 -7280.094,E2 -7280.094} C_VEL
LIN {X 0,Y 474.572,Z 445.412,A -85,B 0,C 180,E1 -7280.841,E2 -7280.841} C_VEL
LIN {X 0,Y 474.341,Z 452.821,A -85,B 0,C 180,E1 -7281.695,E2 -7281.695} C_VEL
LIN {X 0,Y 474.103,Z 460.34,A -85,B 0,C 180,E1 -7282.763,E2 -7282.763} C_VEL
LIN {X 0,Y 473.931,Z 467.219,A -85,B 0,C 180,E1 -7284.043,E2 -7284.043} C_VEL
LIN {X 0,Y 473.792,Z 472.428,A -85,B 0,C 180,E1 -7285.322,E2 -7285.322} C_VEL
LIN {X 0,Y 473.829,Z 475.098,A -85,B 0,C 180,E1 -7286.174,E2 -7286.174} C_VEL
LIN {X 0,Y 473.765,Z 478.016,A -85,B 0,C 180,E1 -7287.45,E2 -7287.45} C_VEL
LIN {X 0,Y 473.755,Z 479.276,A -85,B 0,C 180,E1 -7288.301,E2 -7288.301} C_VEL
LIN {X 0,Y 473.687,Z 480.055,A -85,B 0,C 180,E1 -7289.151,E2 -7289.151} C_VEL
LIN {X 0,Y 473.67,Z 480.342,A -85,B 0,C 180,E1 -7290.001,E2 -7290.001} C_VEL
LIN {X 0,Y 473.687,Z 480.036,A -85,B 0,C 180,E1 -7290.851,E2 -7290.851} C_VEL
LIN {X 0,Y 473.756,Z 479.242,A -85,B 0,C 180,E1 -7291.701,E2 -7291.701} C_VEL
LIN {X 0,Y 473.765,Z 477.966,A -85,B 0,C 180,E1 -7292.552,E2 -7292.552} C_VEL
LIN {X 0,Y 473.828,Z 475.021,A -85,B 0,C 180,E1 -7293.828,E2 -7293.828} C_VEL
LIN {X 0,Y 473.793,Z 472.334,A -85,B 0,C 180,E1 -7294.681,E2 -7294.681} C_VEL
LIN {X 0,Y 473.932,Z 467.092,A -85,B 0,C 180,E1 -7295.959,E2 -7295.959} C_VEL
LIN {X 0,Y 474.125,Z 460.185,A -85,B 0,C 180,E1 -7297.239,E2 -7297.239} C_VEL
LIN {X 0,Y 474.317,Z 452.646,A -85,B 0,C 180,E1 -7298.307,E2 -7298.307} C_VEL
LIN {X 0,Y 474.569,Z 445.224,A -85,B 0,C 180,E1 -7299.161,E2 -7299.161} C_VEL
LIN {X 0,Y 474.848,Z 437.285,A -85,B 0,C 180,E1 -7299.908,E2 -7299.908} C_VEL
LIN {X 0,Y 475.207,Z 427.406,A -85,B 0,C 180,E1 -7300.654,E2 -7300.654} C_VEL
LIN {X 0,Y 475.562,Z 416.823,A -85,B 0,C 180,E1 -7301.251,E2 -7301.251} C_VEL
LIN {X 0,Y 474.784,Z 406.483,A -85,B 0,C 180,E1 -7301.694,E2 -7301.694} C_VEL
LIN {X 0,Y 473.931,Z 398.301,A -85,B 0,C 180,E1 -7301.954,E2 -7301.954} C_VEL
LIN {X 0,Y 474.089,Z 387.919,A -85,B 0,C 180,E1 -7305.512,E2 -7305.512} C_VEL
LIN {X 0,Y 474.299,Z 377.899,A -85,B 0,C 180,E1 -7309.026,E2 -7309.026} C_VEL
LIN {X 0,Y 474.473,Z 370.357,A -85,B 0,C 180,E1 -7311.735,E2 -7311.735} C_VEL
LIN {X 0,Y 474.786,Z 361.627,A -85,B 0,C 180,E1 -7314.954,E2 -7314.954} C_VEL
LIN {X 0,Y 475.078,Z 354.237,A -85,B 0,C 180,E1 -7317.788,E2 -7317.788} C_VEL
LIN {X 0,Y 475.475,Z 347.192,A -85,B 0,C 180,E1 -7320.585,E2 -7320.585} C_VEL
LIN {X 0,Y 475.767,Z 341.04,A -85,B 0,C 180,E1 -7323.132,E2 -7323.132} C_VEL
LIN {X 0,Y 474.784,Z 335.051,A -85,B 0,C 180,E1 -7325.872,E2 -7325.872} C_VEL
LIN {X 0,Y 474.617,Z 334.18,A -85,B 0,C 180,E1 -7326.322,E2 -7326.322} C_VEL
LIN {X 0,Y 474.633,Z 334.181,A -85,B 0,C 180,E1 -7329.648,E2 -7329.648} C_VEL
LIN {X 0,Y 474.621,Z 334.184,A -85,B 0,C 180,E1 -7332.935,E2 -7332.935} C_VEL
LIN {X 0,Y 474.611,Z 334.181,A -85,B 0,C 180,E1 -7335.895,E2 -7335.895} C_VEL
LIN {X 0,Y 474.634,Z 334.177,A -85,B 0,C 180,E1 -7339.041,E2 -7339.041} C_VEL
LIN {X 0,Y 474.615,Z 334.179,A -85,B 0,C 180,E1 -7341.704,E2 -7341.704} C_VEL
LIN {X 0,Y 474.629,Z 334.179,A -85,B 0,C 180,E1 -7344.726,E2 -7344.726} C_VEL
LIN {X 0,Y 474.641,Z 334.176,A -85,B 0,C 180,E1 -7347.788,E2 -7347.788} C_VEL
LIN {X 0,Y 474.628,Z 334.177,A -85,B 0,C 180,E1 -7350.885,E2 -7350.885} C_VEL
LIN {X 0,Y 474.665,Z 334.172,A -85,B 0,C 180,E1 -7353.628,E2 -7353.628} C_VEL
LIN {X 0,Y 474.643,Z 334.176,A -85,B 0,C 180,E1 -7356.641,E2 -7356.641} C_VEL
LIN {X 0,Y 474.66,Z 334.175,A -85,B 0,C 180,E1 -7360.089,E2 -7360.089} C_VEL
LIN {X 0,Y 474.645,Z 334.174,A -85,B 0,C 180,E1 -7362.774,E2 -7362.774} C_VEL
LIN {X 0,Y 474.653,Z 334.174,A -85,B 0,C 180,E1 -7365.42,E2 -7365.42} C_VEL
LIN {X 0,Y 474.711,Z 334.167,A -85,B 0,C 180,E1 -7368.037,E2 -7368.037} C_VEL
LIN {X 0,Y 474.717,Z 334.166,A -85,B 0,C 180,E1 -7371.486,E2 -7371.486} C_VEL
LIN {X 0,Y 474.75,Z 334.162,A -85,B 0,C 180,E1 -7374.903,E2 -7374.903} C_VEL
LIN {X 0,Y 474.89,Z 334.145,A -85,B 0,C 180,E1 -7377.455,E2 -7377.455} C_VEL
LIN {X 0,Y 474.916,Z 334.143,A -85,B 0,C 180,E1 -7379.999,E2 -7379.999} C_VEL
LIN {X 0,Y 474.896,Z 334.145,A -85,B 0,C 180,E1 -7382.544,E2 -7382.544} C_VEL
LIN {X 0,Y 474.777,Z 334.16,A -85,B 0,C 180,E1 -7385.947,E2 -7385.947} C_VEL
LIN {X 0,Y 474.715,Z 334.167,A -85,B 0,C 180,E1 -7388.513,E2 -7388.513} C_VEL
LIN {X 0,Y 474.708,Z 334.17,A -85,B 0,C 180,E1 -7391.961,E2 -7391.961} C_VEL
LIN {X 0,Y 474.703,Z 334.173,A -85,B 0,C 180,E1 -7395.455,E2 -7395.455} C_VEL
LIN {X 0,Y 474.482,Z 334.198,A -85,B 0,C 180,E1 -7398.563,E2 -7398.563} C_VEL
LIN {X 0,Y 474.312,Z 334.722,A -85,B 0,C 180,E1 -7399.924,E2 -7399.924} C_VEL
LIN {X 0,Y 474.185,Z 339.272,A -85,B 0,C 180,E1 -7403.588,E2 -7403.588} C_VEL
LIN {X 0,Y 474.052,Z 342.792,A -85,B 0,C 180,E1 -7406.407,E2 -7406.407} C_VEL
LIN {X 0,Y 473.994,Z 346.473,A -85,B 0,C 180,E1 -7409.293,E2 -7409.293} C_VEL
LIN {X 0,Y 473.906,Z 350.363,A -85,B 0,C 180,E1 -7412.294,E2 -7412.294} C_VEL
LIN {X 0,Y 473.822,Z 354.35,A -85,B 0,C 180,E1 -7415.342,E2 -7415.342} C_VEL
LIN {X 0,Y 473.798,Z 358.234,A -85,B 0,C 180,E1 -7418.162,E2 -7418.162} C_VEL
LIN {X 0,Y 475.635,Z 368.133,A -85,B 0,C 180,E1 -7418.561,E2 -7418.561} C_VEL
LIN {X 0,Y 475.766,Z 375.136,A -85,B 0,C 180,E1 -7418.887,E2 -7418.887} C_VEL
LIN {X 0,Y 475.479,Z 385.706,A -85,B 0,C 180,E1 -7419.533,E2 -7419.533} C_VEL
LIN {X 0,Y 475.18,Z 393.685,A -85,B 0,C 180,E1 -7420.15,E2 -7420.15} C_VEL
LIN {X 0,Y 474.943,Z 400.686,A -85,B 0,C 180,E1 -7420.81,E2 -7420.81} C_VEL
LIN {X 0,Y 474.691,Z 407.387,A -85,B 0,C 180,E1 -7421.568,E2 -7421.568} C_VEL
LIN {X 0,Y 474.519,Z 413.207,A -85,B 0,C 180,E1 -7422.358,E2 -7422.358} C_VEL
LIN {X 0,Y 474.321,Z 418.398,A -85,B 0,C 180,E1 -7423.198,E2 -7423.198} C_VEL
LIN {X 0,Y 474.132,Z 423.285,A -85,B 0,C 180,E1 -7424.159,E2 -7424.159} C_VEL
LIN {X 0,Y 473.972,Z 428.133,A -85,B 0,C 180,E1 -7425.375,E2 -7425.375} C_VEL
LIN {X 0,Y 473.833,Z 431.79,A -85,B 0,C 180,E1 -7426.615,E2 -7426.615} C_VEL
LIN {X 0,Y 473.733,Z 434.58,A -85,B 0,C 180,E1 -7428.118,E2 -7428.118} C_VEL
LIN {X 0,Y 473.711,Z 435.618,A -85,B 0,C 180,E1 -7429.247,E2 -7429.247} C_VEL
LIN {X 0,Y 473.644,Z 435.736,A -85,B 0,C 180,E1 -7430.494,E2 -7430.494} C_VEL
LIN {X 0,Y 473.67,Z 434.68,A -85,B 0,C 180,E1 -7431.846,E2 -7431.846} C_VEL
LIN {X 0,Y 473.79,Z 432.331,A -85,B 0,C 180,E1 -7433.225,E2 -7433.225} C_VEL
LIN {X 0,Y 473.923,Z 428.2,A -85,B 0,C 180,E1 -7434.665,E2 -7434.665} C_VEL
LIN {X 0,Y 474.074,Z 424.118,A -85,B 0,C 180,E1 -7435.712,E2 -7435.712} C_VEL
LIN {X 0,Y 474.244,Z 419.02,A -85,B 0,C 180,E1 -7436.747,E2 -7436.747} C_VEL
LIN {X 0,Y 474.443,Z 413.881,A -85,B 0,C 180,E1 -7437.6,E2 -7437.6} C_VEL
LIN {X 0,Y 474.654,Z 408.007,A -85,B 0,C 180,E1 -7438.413,E2 -7438.413} C_VEL
LIN {X 0,Y 474.904,Z 401.057,A -85,B 0,C 180,E1 -7439.212,E2 -7439.212} C_VEL
LIN {X 0,Y 475.126,Z 393.537,A -85,B 0,C 180,E1 -7439.926,E2 -7439.926} C_VEL
LIN {X 0,Y 475.428,Z 384.48,A -85,B 0,C 180,E1 -7440.621,E2 -7440.621} C_VEL
LIN {X 0,Y 475.761,Z 373.823,A -85,B 0,C 180,E1 -7441.247,E2 -7441.247} C_VEL
LIN {X 0,Y 475.601,Z 367.468,A -85,B 0,C 180,E1 -7441.538,E2 -7441.538} C_VEL
LIN {X 0,Y 475.126,Z 364.933,A -85,B 0,C 180,E1 -7441.651,E2 -7441.651} C_VEL
LIN {X 0,Y 474.134,Z 361.795,A -85,B 0,C 180,E1 -7441.867,E2 -7441.867} C_VEL
LIN {X 0,Y 472.859,Z 359.41,A -85,B 0,C 180,E1 -7442.188,E2 -7442.188} C_VEL
LIN {X 0,Y 470.799,Z 357.012,A -85,B 0,C 180,E1 -7442.79,E2 -7442.79} C_VEL
LIN {X 0,Y 468.859,Z 355.929,A -85,B 0,C 180,E1 -7443.496,E2 -7443.496} C_VEL
LIN {X 0,Y 467.064,Z 354.734,A -85,B 0,C 180,E1 -7444.514,E2 -7444.514} C_VEL
LIN {X 0,Y 466.785,Z 354.038,A -85,B 0,C 180,E1 -7445.033,E2 -7445.033} C_VEL
LIN {X 0,Y 466.797,Z 350.251,A -85,B 0,C 180,E1 -7447.888,E2 -7447.888} C_VEL
LIN {X 0,Y 466.863,Z 346.618,A -85,B 0,C 180,E1 -7450.659,E2 -7450.659} C_VEL
LIN {X 0,Y 466.955,Z 343.082,A -85,B 0,C 180,E1 -7453.383,E2 -7453.383} C_VEL
LIN {X 0,Y 467.007,Z 339.653,A -85,B 0,C 180,E1 -7456.066,E2 -7456.066} C_VEL
LIN {X 0,Y 467.177,Z 336.277,A -85,B 0,C 180,E1 -7458.721,E2 -7458.721} C_VEL
LIN {X 0,Y 467.153,Z 335.183,A -85,B 0,C 180,E1 -7459.598,E2 -7459.598} C_VEL
LIN {X 0,Y 467.671,Z 335.044,A -85,B 0,C 180,E1 -7462.657,E2 -7462.657} C_VEL
LIN {X 0,Y 467.713,Z 335.038,A -85,B 0,C 180,E1 -7464.826,E2 -7464.826} C_VEL
LIN {X 0,Y 467.849,Z 335.022,A -85,B 0,C 180,E1 -7467.416,E2 -7467.416} C_VEL
LIN {X 0,Y 467.871,Z 335.02,A -85,B 0,C 180,E1 -7469.999,E2 -7469.999} C_VEL
LIN {X 0,Y 467.851,Z 335.021,A -85,B 0,C 180,E1 -7472.582,E2 -7472.582} C_VEL
LIN {X 0,Y 467.742,Z 335.036,A -85,B 0,C 180,E1 -7476.036,E2 -7476.036} C_VEL
LIN {X 0,Y 467.671,Z 335.042,A -85,B 0,C 180,E1 -7478.642,E2 -7478.642} C_VEL
LIN {X 0,Y 467.671,Z 335.044,A -85,B 0,C 180,E1 -7482.144,E2 -7482.144} C_VEL
LIN {X 0,Y 467.636,Z 335.048,A -85,B 0,C 180,E1 -7485.885,E2 -7485.885} C_VEL
LIN {X 0,Y 467.611,Z 335.053,A -85,B 0,C 180,E1 -7489.307,E2 -7489.307} C_VEL
LIN {X 0,Y 467.522,Z 335.062,A -85,B 0,C 180,E1 -7492.073,E2 -7492.073} C_VEL
LIN {X 0,Y 467.589,Z 335.053,A -85,B 0,C 180,E1 -7494.887,E2 -7494.887} C_VEL
LIN {X 0,Y 467.614,Z 335.051,A -85,B 0,C 180,E1 -7497.768,E2 -7497.768} C_VEL
LIN {X 0,Y 467.558,Z 335.058,A -85,B 0,C 180,E1 -7501.045,E2 -7501.045} C_VEL
LIN {X 0,Y 467.575,Z 335.054,A -85,B 0,C 180,E1 -7504.242,E2 -7504.242} C_VEL
LIN {X 0,Y 467.538,Z 335.062,A -85,B 0,C 180,E1 -7507.187,E2 -7507.187} C_VEL
LIN {X 0,Y 467.583,Z 335.053,A -85,B 0,C 180,E1 -7510.262,E2 -7510.262} C_VEL
LIN {X 0,Y 467.604,Z 335.052,A -85,B 0,C 180,E1 -7512.571,E2 -7512.571} C_VEL
LIN {X 0,Y 467.559,Z 335.057,A -85,B 0,C 180,E1 -7516.176,E2 -7516.176} C_VEL
LIN {X 0,Y 467.574,Z 335.056,A -85,B 0,C 180,E1 -7518.722,E2 -7518.722} C_VEL
LIN {X 0,Y 467.564,Z 335.057,A -85,B 0,C 180,E1 -7521.406,E2 -7521.406} C_VEL
LIN {X 0,Y 467.549,Z 335.059,A -85,B 0,C 180,E1 -7524.26,E2 -7524.26} C_VEL
LIN {X 0,Y 467.567,Z 335.056,A -85,B 0,C 180,E1 -7527.321,E2 -7527.321} C_VEL
LIN {X 0,Y 467.564,Z 335.058,A -85,B 0,C 180,E1 -7530.666,E2 -7530.666} C_VEL
LIN {X 0,Y 467.602,Z 335.051,A -85,B 0,C 180,E1 -7533.2,E2 -7533.2} C_VEL
LIN {X 0,Y 467.58,Z 335.057,A -85,B 0,C 180,E1 -7536.468,E2 -7536.468} C_VEL
LIN {X 0,Y 467.612,Z 335.05,A -85,B 0,C 180,E1 -7539.778,E2 -7539.778} C_VEL
LIN {X 0,Y 467.596,Z 335.055,A -85,B 0,C 180,E1 -7542.507,E2 -7542.507} C_VEL
LIN {X 0,Y 467.593,Z 335.052,A -85,B 0,C 180,E1 -7545.197,E2 -7545.197} C_VEL
LIN {X 0,Y 467.67,Z 335.044,A -85,B 0,C 180,E1 -7547.856,E2 -7547.856} C_VEL
LIN {X 0,Y 467.67,Z 335.043,A -85,B 0,C 180,E1 -7551.358,E2 -7551.358} C_VEL
LIN {X 0,Y 467.733,Z 335.036,A -85,B 0,C 180,E1 -7553.963,E2 -7553.963} C_VEL
LIN {X 0,Y 467.85,Z 335.022,A -85,B 0,C 180,E1 -7557.418,E2 -7557.418} C_VEL
LIN {X 0,Y 467.87,Z 335.019,A -85,B 0,C 180,E1 -7560.001,E2 -7560.001} C_VEL
LIN {X 0,Y 467.851,Z 335.021,A -85,B 0,C 180,E1 -7562.584,E2 -7562.584} C_VEL
LIN {X 0,Y 467.733,Z 335.036,A -85,B 0,C 180,E1 -7566.038,E2 -7566.038} C_VEL
LIN {X 0,Y 467.672,Z 335.042,A -85,B 0,C 180,E1 -7568.644,E2 -7568.644} C_VEL
LIN {X 0,Y 467.673,Z 335.043,A -85,B 0,C 180,E1 -7572.146,E2 -7572.146} C_VEL
LIN {X 0,Y 467.64,Z 335.048,A -85,B 0,C 180,E1 -7575.886,E2 -7575.886} C_VEL
LIN {X 0,Y 467.614,Z 335.051,A -85,B 0,C 180,E1 -7579.309,E2 -7579.309} C_VEL
LIN {X 0,Y 467.526,Z 335.062,A -85,B 0,C 180,E1 -7582.075,E2 -7582.075} C_VEL
LIN {X 0,Y 467.595,Z 335.053,A -85,B 0,C 180,E1 -7584.888,E2 -7584.888} C_VEL
LIN {X 0,Y 467.62,Z 335.049,A -85,B 0,C 180,E1 -7587.77,E2 -7587.77} C_VEL
LIN {X 0,Y 467.564,Z 335.059,A -85,B 0,C 180,E1 -7591.047,E2 -7591.047} C_VEL
LIN {X 0,Y 467.583,Z 335.053,A -85,B 0,C 180,E1 -7594.244,E2 -7594.244} C_VEL
LIN {X 0,Y 467.543,Z 335.061,A -85,B 0,C 180,E1 -7597.188,E2 -7597.188} C_VEL
LIN {X 0,Y 467.572,Z 335.054,A -85,B 0,C 180,E1 -7600.266,E2 -7600.266} C_VEL
LIN {X 0,Y 467.58,Z 335.055,A -85,B 0,C 180,E1 -7602.568,E2 -7602.568} C_VEL
LIN {X 0,Y 467.565,Z 335.057,A -85,B 0,C 180,E1 -7605.054,E2 -7605.054} C_VEL
LIN {X 0,Y 467.583,Z 335.054,A -85,B 0,C 180,E1 -7607.441,E2 -7607.441} C_VEL
LIN {X 0,Y 467.578,Z 335.055,A -85,B 0,C 180,E1 -7610.857,E2 -7610.857} C_VEL
LIN {X 0,Y 467.592,Z 335.07,A -85,B 0,C 180,E1 -7613.716,E2 -7613.716} C_VEL
LIN {X 0,Y 468.604,Z 340.917,A -85,B 0,C 180,E1 -7616.297,E2 -7616.297} C_VEL
LIN {X 0,Y 468.714,Z 344.594,A -85,B 0,C 180,E1 -7617.841,E2 -7617.841} C_VEL
LIN {X 0,Y 468.302,Z 352.228,A -85,B 0,C 180,E1 -7620.9,E2 -7620.9} C_VEL
LIN {X 0,Y 467.857,Z 361.067,A -85,B 0,C 180,E1 -7624.33,E2 -7624.33} C_VEL
LIN {X 0,Y 467.513,Z 369.381,A -85,B 0,C 180,E1 -7627.461,E2 -7627.461} C_VEL
LIN {X 0,Y 467.242,Z 378.138,A -85,B 0,C 180,E1 -7630.677,E2 -7630.677} C_VEL
LIN {X 0,Y 467.075,Z 386.936,A -85,B 0,C 180,E1 -7633.839,E2 -7633.839} C_VEL
LIN {X 0,Y 466.868,Z 395.711,A -85,B 0,C 180,E1 -7636.951,E2 -7636.951} C_VEL
LIN {X 0,Y 466.849,Z 398.294,A -85,B 0,C 180,E1 -7637.859,E2 -7637.859} C_VEL
LIN {X 0,Y 468.061,Z 410.561,A -85,B 0,C 180,E1 -7638.295,E2 -7638.295} C_VEL
LIN {X 0,Y 468.528,Z 417.176,A -85,B 0,C 180,E1 -7638.606,E2 -7638.606} C_VEL
LIN {X 0,Y 468.27,Z 427.242,A -85,B 0,C 180,E1 -7639.188,E2 -7639.188} C_VEL
LIN {X 0,Y 467.868,Z 437.118,A -85,B 0,C 180,E1 -7639.945,E2 -7639.945} C_VEL
LIN {X 0,Y 467.544,Z 445.046,A -85,B 0,C 180,E1 -7640.702,E2 -7640.702} C_VEL
LIN {X 0,Y 467.302,Z 452.463,A -85,B 0,C 180,E1 -7641.569,E2 -7641.569} C_VEL
LIN {X 0,Y 467.041,Z 459.989,A -85,B 0,C 180,E1 -7642.653,E2 -7642.653} C_VEL
LIN {X 0,Y 466.839,Z 466.876,A -85,B 0,C 180,E1 -7643.952,E2 -7643.952} C_VEL
LIN {X 0,Y 466.72,Z 472.09,A -85,B 0,C 180,E1 -7645.25,E2 -7645.25} C_VEL
LIN {X 0,Y 466.718,Z 474.761,A -85,B 0,C 180,E1 -7646.116,E2 -7646.116} C_VEL
LIN {X 0,Y 466.686,Z 477.683,A -85,B 0,C 180,E1 -7647.412,E2 -7647.412} C_VEL
LIN {X 0,Y 466.661,Z 478.943,A -85,B 0,C 180,E1 -7648.275,E2 -7648.275} C_VEL
LIN {X 0,Y 466.618,Z 479.723,A -85,B 0,C 180,E1 -7649.138,E2 -7649.138} C_VEL
LIN {X 0,Y 466.599,Z 480.01,A -85,B 0,C 180,E1 -7650.001,E2 -7650.001} C_VEL
